# B&R Automation Studio project BenchEDM_AS6
Automation Studio 6.3.2.2; technology packages: mappCockpit 6.2.1, mappConnect 6.1.0, mappControl 6.1.0, mappMotion 6.2.0, mappSafety 6.2.0, mappServices 6.2.0, mappView 6.2.0, OpcUaCs 6.0.0

## Configuration Config1

CPU 5APC3100.KBU2-000, AutomationRuntime 6.3.4, Build 11.3.0, Vc 6.0.0

CPU 5PPC2200.AL04-000, AutomationRuntime 6.3.4, Build 11.3.0, Vc 6.0.0

### Task classes (Cpu.sw)
```
Cyclic#1 (cycle 2000 us, tolerance 0 us):
  Sim <- Process.Sim.prg
  InputMan <- Process.InputMan.prg
  Monitor <- Process.Monitor.prg
  Seq_MASTER <- Process.Seq_MASTER.prg
  OutputMan <- Process.OutputMan.prg
Cyclic#8 (cycle 2000 us):
  BuildVer <- BuildVersion.BuildVer.prg
  Services <- Services.prg
  Vis <- Vis.prg
  Dev <- Dev.prg
DataObjects: MbRTU <- Libraries.MbRTU.dob, McAcpSys, datamod
NcDataObjects: AcpParTabL <- Libraries.AcpParTabL.dob, McDriveLog
Binaries: udbdef, mvLoader, TCLang, TCData, FWRules, ArSvcReg, mvConfig, McAcpSim, McAcpDrv, McMechSys, mvDatApi, McProfGen, BRRole, iomap, asfw, Role, ashwac, UaCsConfig, sysconf, TC, ashwd, User, arconfig, AlarmHist, Config, AlarmCore, AlarmList, Config_1, mCoWebSc, Settings, Config_2, Hierarchy, Config_3, Config_4, Config_6, asnxdb1, Config_5, AlarmCat
ReActionTechnologyObjects: StepDir <- StepDir.prg
Libraries: TC_General, TC_Version, TC_IO, TC_Dir, TC_Convert, TC_ItemX, TC_Array, TC_SysErr, TC_Eval, TC_Mon, TC_Recipe, TC_Sim, TC_AlarmX, TC_RAND, operator, runtime, AsIecCon, astime, ArEventLog, ArProject, AsBrStr, brsystem, FileIO, AsUSB, standard, ArTextSys, sys_lib, MTTypes, MTBasics, MTFilter, AsSMTP, ArCert, ArSsl, AsIODiag, AsTCP, AsXml, MpAlarmX, MpBase, MpRecipe, McBase, MpAxis, McAxis, McAcpAx, AsZip, McAxGroup, McPathGen, McProgInt, SfDomain, MpCnc, McPureVAx, AsIORTI, TC_Str, CoTrace, DRV_mbus, dvframe, DataObj, HA_Matrix, TC_NGRC, TC_Seq, TC_JSON, AsBrMath, TC_FrSky, AsUDP, UaCoal, UaCoalPrv, powerlnk, AsEPL, SfDomDrv, AsIO, AsMem, AsIOAcc, ArUser, MpSfDomMgr, SfDomVis, AsArProf
```

### Hardware
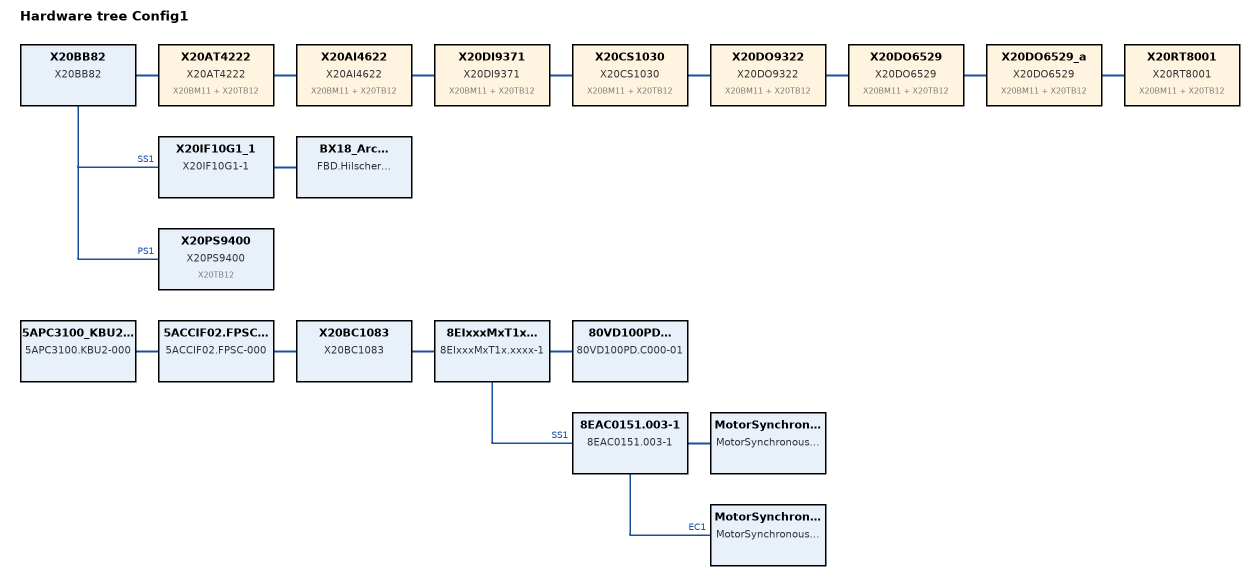
```
5ACCIF02.FPSC-000_a : 5ACCIF02.FPSC-000 v1.6.0.0  [SL -> 5APC3100_KBU2_000_a.SL2]
  Connector IF1:
    EplNatSubnet = 192.168.102.0
    Channel1
    ChannelID1 = McAcpBroadcast
    ChannelType1 = OCTET[96]
  Supervision = off
5APC3100_KBU2_000_a : 5APC3100.KBU2-000 v2.3.0.0
  Connector IF3:
    AssignedOperatingSystem = GPOS
  Connector IF4:
    AssignedOperatingSystem = ARemb
    ActivateDevice = 1
    Mode = Manual
    InternetAddress = 192.168.0.2
    SubnetMask = 255.255.255.0
    ActivateSnmp = 2
  Connector IF9:
    OperatingSystem = ARemb
    ActivateDevice = 1
  Connector IF5:
    AssignedOperatingSystem = GPOS
  Connector IF6:
    AssignedOperatingSystem = GPOS
  Connector IF7:
    AssignedOperatingSystem = ARemb
  Connector IF8:
    AssignedOperatingSystem = ARemb
  ConfigurationID = Config1
  UserPartitionSize = 10000
  UserRamDevice = PCI.2.FPSC.SRAM
  UserRamSize = 14000
  RemMemDevice = PCI.2.FPSC.SRAM
  RemMemSize = 200000
  RemanentGlobalPvSize = 200000
  VolatileGlobalPvSize = 6553500
  ClearNvMemoryAfterShutdownFlushError = 0
  CyclicFlushRemMemSelector = 1
  CyclicFlushRemMemCycleTime = 300
  EnableUsbRemoteInstall = 1
  TimerDeviceType = EPLX2X
  TimerDevice = 5ACCIF02.FPSC-000_a.IF1
  TaskClassIdleTime = 10000
  Cyclic1Duration = 2000
  Cyclic1Tolerance = 0
  Cyclic1Stack = 655360
  Cyclic1Output = 1
  Cyclic8Duration = 2000
  FileDevice1
  FileDeviceName1 = USER_DEVICE
  FileDevicePath1 = F:\
  FileDevice2
  FileDeviceName2 = USER_DEVICE_SIM
  FileDevicePath2 = ..\..\..\..\USER_DEVICE\
  EthernetDefaultGateway = 192.168.0.1
  ActivateFtpServer = 1
  FTPProtocol = 1
  FtpUser1
  FtpUsername1 = brcpu
  FtpUserPassword1 = Ga9FbfaYwFdrzzlreMI/KhLrdRli8oqxPKsqgG5NU/A=
  FtpUserSalt1 = BqJHaXjm
  FTPAccessRight1 = 0
  FTPdevice1 = ALL
  ActivateWebServer = 1
  WebServerProtocol = 1
  ActivateSdm = 1
  ActivateHypervisor = 1
  ARembDramSizeInMb = 3072
80VD100PD.C000-01 : 80VD100PD.C000-01 v2.5.1.0 (NodeNumber=3)  [PLK1 -> 8EIxxxMxT1x.xxxx-1.PLK2 [Cable Type=PowerlinkCable, Length=10, Version=1.0.0.3]]
  DriveConfiguration/Channel[1]/RealAxis:
    AxisReference = gAxisRV_0_0
  DriveConfiguration/Channel[1]/RealAxis/MechanicalElements/Gearbox:
    Input = 10
  DriveConfiguration/Channel[1]/RealAxis/Controller/Mode/Position:
    IntegrationTime = 0.05
  DriveConfiguration/Channel[1]/RealAxis/Controller/Mode/Speed:
    ProportionalGain = 0.2
  DriveConfiguration/Channel[1]/RealAxis/MovementErrorLimits:
    VelocityErrorMonitoring = NotUsed
  DriveConfiguration/Channel[1]/RealAxis/DigitalInputs/Quickstop:
    Input = NotUsed
  DriveConfiguration/Channel[1]/ChannelFeatures:
    FeatureRef[1] = Feature_AcpParTable
  DriveConfiguration/Channel[2]/RealAxis:
    AxisReference = gAxisRT_0_0
  DriveConfiguration/Channel[2]/RealAxis/Controller/Mode/Position:
    ProportionalGain = 500
    IntegrationTime = 0.01
    PredictionTime = 0.003
    TotalDelayTime = 0.003
  DriveConfiguration/Channel[2]/RealAxis/Controller/Mode/Speed:
    ProportionalGain = 0.05
  DriveConfiguration/Channel[2]/RealAxis/MovementErrorLimits:
    VelocityErrorMonitoring = NotUsed
  DriveConfiguration/Channel[2]/RealAxis/DigitalInputs/Quickstop:
    Input = NotUsed
  DriveConfiguration/Channel[2]/ChannelFeatures:
    FeatureRef[1] = Feature_AcpParTable
8EAC0151.003-1 : 8EAC0151.003-1 v2.2.1.0  [SS -> 8EIxxxMxT1x.xxxx-1.SS1; EC1 -> MotorSynchronous_any_a.EC; EC2 -> MotorSynchronous_any.EC]
  Encoder/EncoderX41x:
    InterfaceType = IncrementalEAC151
  Encoder/EncoderX41x/InterfaceType/PowerSupply:
    ReferencePulseDetection = 512
    LineCount = 5000
  Encoder/EncoderX42x:
    InterfaceType = IncrementalEAC151
  Encoder/EncoderX42x/InterfaceType/PowerSupply:
    ReferencePulseDetection = 512
    LineCount = 5000
8EIxxxMxT1x.xxxx-1 : 8EIxxxMxT1x.xxxx-1 v2.4.0.0 (NodeNumber=2)  [PLK1 -> X20BC1083.PLK2 [Cable Type=PowerlinkCable, Length=10, Version=1.0.0.3]; PLK2 -> 80VD100PD.C000-01.PLK1 [Cable Type=PowerlinkCable, Length=10, Version=1.0.0.3]; MT2 -> MotorSynchronous_any.MT]
  PDMConfig = DoubleAxis
  DriveConfiguration/Encoder/EncoderX43:
    InterfaceType = EnDat
  DriveConfiguration/Channel[1]/RealAxis:
    AxisReference = gAxisRY_0_0
  DriveConfiguration/Channel[1]/RealAxis/MechanicalElements/RotaryToLinearTransformation:
    ReferenceDistance = 20
  DriveConfiguration/Channel[1]/RealAxis/EncoderLink:
    MotorAndPositionEncoder = EncoderX41x
  DriveConfiguration/Channel[1]/RealAxis/Controller:
    Mode = PositionControllerWithTorqueFeedForward
  DriveConfiguration/Channel[1]/RealAxis/Controller/Mode/Position:
    ProportionalGain = 500
    IntegrationTime = 0.1
  DriveConfiguration/Channel[1]/RealAxis/Controller/Mode/Speed:
    ProportionalGain = 0.5
  DriveConfiguration/Channel[1]/RealAxis/Controller/Mode/FeedForward:
    TorquePositive = 0.2
    TorqueNegative = 0.2
    SpeedTorqueFactor = 0.005
    Inertia = 0.00015
  DriveConfiguration/Channel[1]/RealAxis/Homing:
    Mode = BlockTorque
  DriveConfiguration/Channel[1]/RealAxis/Homing/Mode:
    Position = -20
    StartVelocity = 20
    HomingVelocity = 20
    Acceleration = 1000
    StartDirection = Negative
    TorqueLimit = 1.5
    PositionErrorStopLimit = 4
  DriveConfiguration/Channel[1]/RealAxis/MovementErrorLimits:
    PositionError = 5
    VelocityErrorMonitoring = NotUsed
  DriveConfiguration/Channel[1]/ChannelFeatures:
    FeatureRef[1] = Feature_AcpParTable
  DriveConfiguration/Channel[2]/RealAxis:
    AxisReference = gAxisRX_0_0
  DriveConfiguration/Channel[2]/RealAxis/MechanicalElements/RotaryToLinearTransformation:
    ReferenceDistance = 20
  DriveConfiguration/Channel[2]/RealAxis/EncoderLink:
    MotorAndPositionEncoder = EncoderX42x
  DriveConfiguration/Channel[2]/RealAxis/Controller/Mode/Position:
    ProportionalGain = 500
    IntegrationTime = 0.1
  DriveConfiguration/Channel[2]/RealAxis/Controller/Mode/Speed:
    ProportionalGain = 0.5
  DriveConfiguration/Channel[2]/RealAxis/Homing:
    Mode = BlockTorque
  DriveConfiguration/Channel[2]/RealAxis/Homing/Mode:
    Position = -10
    StartVelocity = 20
    HomingVelocity = 20
    Acceleration = 1000
    StartDirection = Negative
    TorqueLimit = 1.5
    PositionErrorStopLimit = 4
  DriveConfiguration/Channel[2]/RealAxis/MovementErrorLimits:
    PositionError = 5
    VelocityErrorMonitoring = NotUsed
  DriveConfiguration/Channel[2]/ChannelFeatures:
    FeatureRef[1] = Feature_AcpParTable
  DriveConfiguration/Channel[3]/RealAxis:
    AxisReference = 
BX18_Arc_Generator_V1_0 : FBD.Hilscher.ECATGenSlaveDTM.BX18 Arc Generator V1.0 v1.0 (OrderNumber=BX18 Arc Generator V1.0)  [ECAT1 -> X20IF10G1_1.IF1]
  DtmId = 61a48d3a-efc3-4167-a8a5-4e7e0e28ba40
MotorSynchronous_any : MotorSynchronous_any v2.2.1.0  [EC -> 8EAC0151.003-1.EC2; MT -> 8EIxxxMxT1x.xxxx-1.MT2]
  M1/MotorParameters:
    MOTOR_POLEPAIRS = 1
    MOTOR_SPEED_RATED = 3300
    MOTOR_SPEED_MAX = 9300
    MOTOR_VOLTAGE_RATED = 300
    MOTOR_CURR_RATED = 2
    MOTOR_CURR_STALL = 2
    MOTOR_CURR_MAX = 8
    MOTOR_TORQ_RATED = 0.66
    MOTOR_TORQ_STALL = 2.55
    MOTOR_TORQ_MAX = 2.65
    MOTOR_VOLTAGE_CONST = 10.53
    MOTOR_TORQ_CONST = 0.302
    MOTOR_STATOR_RESISTANCE = 1.3
    MOTOR_STATOR_INDUCTANCE = 3.8
    MOTOR_INERTIA = 0.172
  M1/MotorParameters/EncoderMounting:
    Angle = Undefined
  M1/MotorParameters/EncoderMounting/Angle:
    AutomaticIdentification = Dither
  M1/MotorParameters/EncoderMounting/Angle/AutomaticIdentification:
    PHASING_CURR = 1.5 (Disabled=false)
  M1/MotorParameters:
    TemperatureSensor = NotUsed
    TemperatureModel = NotUsed
MotorSynchronous_any_a : MotorSynchronous_any v2.2.1.0  [EC -> 8EAC0151.003-1.EC1; MT -> 8EIxxxMxT1x.xxxx-1.MT1]
  M1/MotorParameters:
    MOTOR_POLEPAIRS = 1
    MOTOR_SPEED_RATED = 3300
    MOTOR_SPEED_MAX = 9300
    MOTOR_VOLTAGE_RATED = 300
    MOTOR_CURR_RATED = 2
    MOTOR_CURR_STALL = 2
    MOTOR_CURR_MAX = 8
    MOTOR_TORQ_RATED = 0.66
    MOTOR_TORQ_STALL = 2.55
    MOTOR_TORQ_MAX = 2.65
    MOTOR_VOLTAGE_CONST = 10.53
    MOTOR_TORQ_CONST = 0.302
    MOTOR_STATOR_RESISTANCE = 1.3
    MOTOR_STATOR_INDUCTANCE = 3.8
    MOTOR_INERTIA = 0.172
  M1/MotorParameters/EncoderMounting:
    Angle = Undefined
  M1/MotorParameters/EncoderMounting/Angle:
    AutomaticIdentification = Dither
  M1/MotorParameters/EncoderMounting/Angle/AutomaticIdentification:
    PHASING_CURR = 1.5 (Disabled=false)
  M1/MotorParameters:
    TemperatureSensor = NotUsed
    TemperatureModel = NotUsed
X20AI4622 : X20AI4622 v1.5.0.0  [SS1 -> X20TB12_c.SS; SL -> X20BM11_b.SL1]
  Supervision = off
  ChannelType01 = 0 to 20mA
  ChannelType02 = 0 to 20mA
  ChannelType03 = 0 to 20mA
  ChannelType04 = 0 to 20mA
X20AT4222 : X20AT4222 v1.6.2.0  [SS1 -> X20TB12.SS; SL -> X20BM11_a.SL1]
  Supervision = off
X20BB82 : X20BB82 v1.2.0.0
X20BC1083 : X20BC1083 v2.16.1.0 (NodeNumber=1)  [PLK1 -> 5ACCIF02.FPSC-000_a.IF1 [Cable Type=PowerlinkCable, Length=10, Version=1.0.0.3]; PLK2 -> 8EIxxxMxT1x.xxxx-1.PLK1 [Cable Type=PowerlinkCable, Length=10, Version=1.0.0.3]; SL -> X20BB82.SL1]
  Supervision = off
X20BM11 : X20BM11 v1.1.0.0  [X2X1 -> X20BM11_g.X2X2]
X20BM11_a : X20BM11 v1.1.0.0  [X2X1 -> X20BB82.IF1]
X20BM11_b : X20BM11 v1.1.0.0  [X2X1 -> X20BM11_a.X2X2]
X20BM11_c : X20BM11 v1.1.0.0  [X2X1 -> X20BM11_b.X2X2]
X20BM11_d : X20BM11 v1.1.0.0  [X2X1 -> X20BM11_c.X2X2]
X20BM11_e : X20BM11 v1.1.0.0  [X2X1 -> X20BM11_d.X2X2]
X20BM11_f : X20BM11 v1.1.0.0  [X2X1 -> X20BM11_e.X2X2]
X20BM11_g : X20BM11 v1.1.0.0  [X2X1 -> X20BM11_f.X2X2]
X20CS1030 : X20CS1030 v1.8.3.0  [SS1 -> X20TB12_e.SS; SL -> X20BM11_d.SL1]
  Supervision = off
X20DI9371 : X20DI9371 v1.6.1.0  [SS1 -> X20TB12_d.SS; SL -> X20BM11_c.SL1]
  Supervision = off
X20DO6529 : X20DO6529 v1.4.1.0  [SS1 -> X20TB12_g.SS; SL -> X20BM11_f.SL1]
  Supervision = off
X20DO6529_a : X20DO6529 v1.4.1.0  [SS1 -> X20TB12_h.SS; SL -> X20BM11_g.SL1]
  Supervision = off
X20DO9322 : X20DO9322 v1.7.0.0  [SS1 -> X20TB12_f.SS; SL -> X20BM11_e.SL1]
  Supervision = off
X20IF10G1_1 : X20IF10G1-1 v1.0.2.0  [SS -> X20BB82.SS1]
  Connector IF1:
    DtmRef = FBDIF.Hilscher.ECATMasterDTM.NETX 100 RE/ECM
    DtmId = 2adc853f-087f-4c82-9441-944b4b0f2f89
  ConfigFile = X20IF10G1_1.dtm
  ConfigModule = asnxdb1
  CycleTime = 2000
X20PS9400 : X20PS9400 v1.8.1.0  [SS1 -> X20TB12_b.SS; PS -> X20BB82.PS1]
  Supervision = off
X20RT8001 : X20RT8001 v1.7.2.0  [SS1 -> X20TB12_a.SS; SL -> X20BM11.SL1]
  Supervision = off
  ReActionTask = StepDir
  ReActionTaskDisabled = FALSE
  TypePar1 = DINT
  TypePar2 = DINT
  TypePar3 = DINT
  TypeRes1 = DINT
X20TB12 : X20TB12 v1.0.0.0
X20TB12_a : X20TB12 v1.0.0.0
X20TB12_b : X20TB12 v1.0.0.0
X20TB12_c : X20TB12 v1.0.0.0
X20TB12_d : X20TB12 v1.0.0.0
X20TB12_e : X20TB12 v1.0.0.0
X20TB12_f : X20TB12 v1.0.0.0
X20TB12_g : X20TB12 v1.0.0.0
X20TB12_h : X20TB12 v1.0.0.0
```

### IoMap.iom - 5APC3100_KBU2_000_a/IoMap.iom
```iecst
VAR_CONFIG
	Cyclic#1.gIO.BX18.Outputs_control AT %QW."BX18_Arc_Generator_V1_0".Outputs_control;
	Cyclic#1.gIO.BX18.Outputs_onTime AT %QW."BX18_Arc_Generator_V1_0".Outputs_onTime;
	Cyclic#1.gIO.BX18.Outputs_offTime AT %QW."BX18_Arc_Generator_V1_0".Outputs_offTime;
	Cyclic#1.gIO.BX18.Outputs_current AT %QW."BX18_Arc_Generator_V1_0".Outputs_current;
	Cyclic#1.gIO.BX18.Inputs_status AT %IW."BX18_Arc_Generator_V1_0".Inputs_status;
	Cyclic#1.gIO.BX18.Inputs_EDMservofeedback AT %IW."BX18_Arc_Generator_V1_0".Inputs_EDMservofeedback;
	Cyclic#1.gIO.BX18.Inputs_power AT %IW."BX18_Arc_Generator_V1_0".Inputs_power;
	Cyclic#1.gIO.BX18.ModuleOK AT %IX."BX18_Arc_Generator_V1_0".ModuleOk;
	Cyclic#1.::gIO.Motion.ModuleOK AT %IX."X20RT8001".ModuleOk;
	Cyclic#1.::gIO.Motion.ENABLED AT %IX."X20RT8001".RTEngineRun;
	Cyclic#1.::gIO.Motion.ActualPosition AT %ID."X20RT8001".RES01;
	Cyclic#1.::gIO.Motion.SetPosition AT %QD."X20RT8001".PAR01;
	Cyclic#1.::gIO.Motion.Home AT %QD."X20RT8001".PAR02;
	Cyclic#1.::gIO.Motion.ENABLE AT %QX."X20RT8001".RTEnable;
	Cyclic#1.::gIO.Safety.TC_IO_DI_ESTOP.IOMapping AT %IX."X20DI9371".DigitalInput01;
	Cyclic#1.::gIO.Motion.StepDelay AT %QD."X20RT8001".PAR03;
	Cyclic#1.::gIO.Motion.TC_IO_DI_HomeSwitchZ.IOMapping AT %IX."X20DI9371".DigitalInput03;
END_VAR
```

### Config.mappconnect - 5APC3100_KBU2_000_a/mappConnect/Config.mappconnect
```
Element mapp Connect Configuration (Type=mappconnect)
  WebServerProtocol = 1
    WebServerPort = 8081
    Interface = All
    WebServerPortSsl = 8443
  WebServerEndpointConfiguration:
    Endpoint[1]:
      Endpoint = *.*
      Roles
  OpcUaServerWhitelist:
    OpcUaServer[1]:
      Url = opc.tcp://127.0.0.1:4840
```

### Config_1.axesgroup - 5APC3100_KBU2_000_a/mappMotion/CNC/Config_1.axesgroup
```
Element gCNC (Type=axesgroup)
  Type = PathGenAxesGroup
    PhysicalAxes:
      JointAxes:
        JointAxis[1]:
          Name = QX
          AxisRef = gAxisVX_0
        JointAxis[2]:
          Name = QY
          AxisRef = gAxisVY_0
        JointAxis[3]:
          Name = QZ
          AxisRef = gAxisVZ_0
    MechanicalSystem:
      MechSysRef = MechSys
    AxesGroupFeatures:
      FeatureRef[1] = Feature_Programs
      FeatureRef[2] = Feature_ReverseMovement
  Alarms = MpAlarmX
```

### Config_2.axis - 5APC3100_KBU2_000_a/mappMotion/CNC/Config_2.axis
```
Element gAxisRP_1_0 (Type=axis)
  BaseType:
    MeasurementUnit = 5059636
    MeasurementResolution = 0.001
    PeriodSettings:
      Period = 1
  MovementLimits:
    Velocity:
      Velocity = 60
    Acceleration:
      Acceleration = 600
    Deceleration:
      Deceleration = 600
  Alarms = MpAlarmX
Element gAxisRP_0_0 (Type=axis)
  BaseType:
    MeasurementUnit = 5059636
    MeasurementResolution = 0.001
    PeriodSettings:
      Period = 1
  MovementLimits:
    Velocity:
      Velocity = 60
    Acceleration:
      Acceleration = 600
    Deceleration:
      Deceleration = 600
  Alarms = MpAlarmX
Element gAxisRT_0_0 (Type=axis)
  BaseType:
    MeasurementResolution = 0.001
  MovementLimits:
    Velocity:
      Velocity = 12000
    Acceleration:
      Acceleration = 120000
    Deceleration:
      Deceleration = 120000
  Alarms = MpAlarmX
Element gAxisRV_0_0 (Type=axis)
  BaseType:
    MeasurementResolution = 0.001
  MovementLimits:
    Velocity:
      Velocity = 1200
    Acceleration:
      Acceleration = 12000
    Deceleration:
      Deceleration = 12000
  Alarms = MpAlarmX
Element gAxisRX_0_0 (Type=axis)
  BaseType = LinearBounded
    MeasurementResolution = 0.001
  MovementLimits:
    Position:
      LowerLimit = 0
      UpperLimit = 250
    Velocity:
      Velocity = 1000
    Acceleration:
      Acceleration = 5000
    Deceleration:
      Deceleration = 5000
  Alarms = MpAlarmX
Element gAxisRY_0_0 (Type=axis)
  BaseType = LinearBounded
    MeasurementResolution = 0.001
  MovementLimits:
    Position:
      LowerLimit = 0
      UpperLimit = 550
    Velocity:
      Velocity = 1000
    Acceleration:
      Acceleration = 5000
    Deceleration:
      Deceleration = 5000
  Alarms = MpAlarmX
Element gAxisRZ_0_0 (Type=axis)
  BaseType = LinearBounded
    MeasurementResolution = 0.001
  MovementLimits:
    Position:
      LowerLimit = 0
      UpperLimit = 265
    Velocity:
      Velocity = 120
    Acceleration:
      Acceleration = 12000
    Deceleration:
      Deceleration = 12000
  Alarms = MpAlarmX
Element gAxisVT_0 (Type=axis)
  BaseType:
    MeasurementResolution = 0.001
  MovementLimits:
    Velocity:
      Velocity = 10000
    Acceleration:
      Acceleration = 100000
    Deceleration:
      Deceleration = 100000
  Alarms = MpAlarmX
Element gAxisVV_0 (Type=axis)
  BaseType:
    MeasurementResolution = 0.001
  MovementLimits:
    Velocity:
      Velocity = 1000
    Acceleration:
      Acceleration = 10000
    Deceleration:
      Deceleration = 10000
  Alarms = MpAlarmX
Element gAxisVX_0 (Type=axis)
  BaseType = LinearBounded
    MeasurementResolution = 0.001
  MovementLimits:
    Position:
      LowerLimit = 0
      UpperLimit = 250
    Velocity:
      Velocity = 800
    Acceleration:
      Acceleration = 4000
    Deceleration:
      Deceleration = 4000
  Alarms = MpAlarmX
Element gAxisVY_0 (Type=axis)
  BaseType = LinearBounded
    MeasurementResolution = 0.001
  MovementLimits:
    Position:
      LowerLimit = 0
      UpperLimit = 550
    Velocity:
      Velocity = 800
    Acceleration:
      Acceleration = 4000
    Deceleration:
      Deceleration = 4000
  Alarms = MpAlarmX
Element gAxisVZ_0 (Type=axis)
  BaseType = LinearBounded
    MeasurementResolution = 0.001
  MovementLimits:
    Position:
      LowerLimit = 0
      UpperLimit = 265
    Velocity:
      Velocity = 100
    Acceleration:
      Acceleration = 10000
    Deceleration:
      Deceleration = 10000
  Alarms = MpAlarmX
```

### Config_3.mechanicalsystem - 5APC3100_KBU2_000_a/mappMotion/CNC/Config_3.mechanicalsystem
```
Element MechSys (Type=mechanicalsystem)
  Type = 3AxesCNC
    Subtype:
      JointAxesPositionLimits:
        JointAxis[1]
        JointAxis[2]
        JointAxis[3]
```

### Config_4.axesgroupfeature - 5APC3100_KBU2_000_a/mappMotion/CNC/Config_4.axesgroupfeature
```
Element Feature_Programs (Type=axesgroupfeature)
  Type:
    Location = User
      UserLocation[1]:
        FileDevice = USER_DEVICE
      UserLocation[2]:
        FileDevice = USER_DEVICE_SIM
Element Feature_ReverseMovement (Type=axesgroupfeature)
  Type = ReverseMovement
    Distance = 5
```

### Config_5.purevaxcfg - 5APC3100_KBU2_000_a/mappMotion/CNC/Config_5.purevaxcfg
```
Element PureVAxCfg_VT_0 (Type=purevaxcfg)
  PureVAxis:
    AxisReference = gAxisVT_0
Element PureVAxCfg_VV_0 (Type=purevaxcfg)
  PureVAxis:
    AxisReference = gAxisVV_0
Element PureVAxCfg_RZ_0_0 (Type=purevaxcfg)
  PureVAxis:
    AxisReference = gAxisRZ_0_0
    Homing:
      Mode = LimitSwitch
        Position = -5
        StartVelocity = 20
        HomingVelocity = 5
        Acceleration = 12000
        SwitchEdge = Negative
    GeneralPurposeAxisInterface = Used
      MovementErrorLimits:
        PositionError = 1000
      DigitalInputs:
        NegativeLimitSwitch:
          Source = InputPV
            PVmapping = gIO.Motion.TC_IO_DI_HomeSwitchZ.Signal.Filtered
        Trigger1:
          Source = InputPV
            PVmapping = ::gIO.Safety.TC_IO_DI_ESTOP.Signal.Filtered
          Level = Low
        Quickstop:
          Input = Trigger1
      StatusInputs:
        PoweredOn:
          Source = InputPV
            PVmapping = ::gIO.Motion.SwitchedOn
        ReadyForPowerOn:
          Source = InputPV
            PVmapping = ::gIO.Motion.ENABLED
      ControlOutputs:
        PowerOn = Used
          Destination:
            PVmapping = ::gIO.Motion.SwitchOn
Element PureVAxCfg_VZ_0 (Type=purevaxcfg)
  PureVAxis:
    AxisReference = gAxisVZ_0
Element PureVAxCfg_VY_0 (Type=purevaxcfg)
  PureVAxis:
    AxisReference = gAxisVY_0
Element PureVAxCfg_VX_0 (Type=purevaxcfg)
  PureVAxis:
    AxisReference = gAxisVX_0
Element PureVAxCfg_RP_1_0 (Type=purevaxcfg)
  PureVAxis:
    AxisReference = gAxisRP_1_0
    GeneralPurposeAxisInterface = DS402VL
      MovementErrorLimits:
        PositionError = 10
      VelocityActualValue:
        Source = Variable
          PVMapping = ::gIO.VFD[1].RFRD
      StatusInputs:
        StatusWord:
          Source = InputPV
            PVmapping = ::gIO.VFD[1].ETA
      ControlOutputs:
        ControlWord:
          Destination:
            PVMapping = ::gIO.VFD[1].CMD
        TargetVelocity:
          Destination:
            PVmapping = ::gIO.VFD[1].LFRD
Element PureVAxCfg_RP_0_0 (Type=purevaxcfg)
  PureVAxis:
    AxisReference = gAxisRP_0_0
    GeneralPurposeAxisInterface = DS402VL
      MovementErrorLimits:
        PositionError = 10
      VelocityActualValue:
        Source = Variable
          PVMapping = ::gIO.VFD[0].RFRD
      StatusInputs:
        StatusWord:
          Source = InputPV
            PVmapping = ::gIO.VFD[0].ETA
      ControlOutputs:
        ControlWord:
          Destination:
            PVMapping = ::gIO.VFD[0].CMD
        TargetVelocity:
          Destination:
            PVmapping = ::gIO.VFD[0].LFRD
```

### Config_6.axisfeature - 5APC3100_KBU2_000_a/mappMotion/CNC/Config_6.axisfeature
```
Element Feature_AcpParTable (Type=axisfeature)
  Type = ParTab
    ParTabRef = AcpParTabL
```

### AlarmList.mpalarmxlist - 5APC3100_KBU2_000_a/mappServices/AlarmList.mpalarmxlist
```
Element gAlarmXList_Base (Type=mpalarmxlist)
  mapp.AlarmX.Core.Configuration:
    [0]:
      Name = {1}Severity0
      Message = {$IAT/Alarm.{1}Severity}
      Code = 0
      Severity = 0
      Behavior = EdgeAlarm
        Confirm = 0
        ReactionWhilePending = TRUE
        Retain = FALSE
        Async = FALSE
        DataUpdate:
          Activation:
            TimeStamp = FALSE
            Snippets = FALSE
        Recording:
          InactiveToActive = TRUE
          UnacknowledgedToAcknowledged = FALSE
          AcknowledgedToUnacknowledged = FALSE
          UnconfirmedToConfirmed = FALSE
          ConfirmedToUnconfirmed = FALSE
      Disable = FALSE
      InhibitPV
      AdditionalInformation1
      AdditionalInformation2
    [1]:
      Name = {1}Severity1
      Message = {$IAT/Alarm.{1}Severity}
      Code = 1
      Severity = 1
      Behavior = EdgeAlarm
        Confirm = 0
        ReactionWhilePending = TRUE
        Retain = FALSE
        Async = FALSE
        DataUpdate:
          Activation:
            TimeStamp = FALSE
            Snippets = FALSE
        Recording:
          InactiveToActive = TRUE
          UnacknowledgedToAcknowledged = FALSE
          AcknowledgedToUnacknowledged = FALSE
          UnconfirmedToConfirmed = FALSE
          ConfirmedToUnconfirmed = FALSE
      Disable = FALSE
      InhibitPV
      AdditionalInformation1
      AdditionalInformation2
    [2]:
      Name = {1}Severity2
      Message = {$IAT/Alarm.{1}Severity}
      Code = 2
      Severity = 2
      Behavior = EdgeAlarm
        Confirm = 0
        ReactionWhilePending = TRUE
        Retain = FALSE
        Async = FALSE
        DataUpdate:
          Activation:
            TimeStamp = FALSE
            Snippets = FALSE
        Recording:
          InactiveToActive = TRUE
          UnacknowledgedToAcknowledged = FALSE
          AcknowledgedToUnacknowledged = FALSE
          UnconfirmedToConfirmed = FALSE
          ConfirmedToUnconfirmed = FALSE
      Disable = FALSE
      InhibitPV
      AdditionalInformation1
      AdditionalInformation2
    [3]:
      Name = {1}Severity3
      Message = {$IAT/Alarm.{1}Severity}
      Code = 3
      Severity = 3
      Behavior = EdgeAlarm
        Confirm = 0
        ReactionWhilePending = TRUE
        Retain = FALSE
        Async = FALSE
        DataUpdate:
          Activation:
            TimeStamp = FALSE
            Snippets = FALSE
        Recording:
          InactiveToActive = TRUE
          UnacknowledgedToAcknowledged = FALSE
          AcknowledgedToUnacknowledged = FALSE
          UnconfirmedToConfirmed = FALSE
          ConfirmedToUnconfirmed = FALSE
      Disable = FALSE
      InhibitPV
      AdditionalInformation1
      AdditionalInformation2
    [4]:
      Name = {1}Severity4
      Message = {$IAT/Alarm.{1}Severity}
      Code = 4
      Severity = 4
      Behavior = EdgeAlarm
        Confirm = 0
        ReactionWhilePending = TRUE
        Retain = FALSE
        Async = FALSE
        DataUpdate:
          Activation:
            TimeStamp = FALSE
            Snippets = FALSE
        Recording:
          InactiveToActive = TRUE
          UnacknowledgedToAcknowledged = FALSE
          AcknowledgedToUnacknowledged = FALSE
          UnconfirmedToConfirmed = FALSE
          ConfirmedToUnconfirmed = FALSE
      Disable = FALSE
      InhibitPV
      AdditionalInformation1
      AdditionalInformation2
  mapp.AlarmX.Snippets:
    AutoDetect = 1
      Language
    [0]:
      Key = TestKey
      Value = PV
        PV = ::gRem.RuntimeHours
      Alarm
```

### Config_1.axesgroup - 5PPC2200_AL04_000/mappMotion/CNC/Config_1.axesgroup
```
Element gCNC (Type=axesgroup)
  Type = PathGenAxesGroup
    PhysicalAxes:
      JointAxes:
        JointAxis[1]:
          Name = QX
          AxisRef = gAxisVX_0
        JointAxis[2]:
          Name = QY
          AxisRef = gAxisVY_0
        JointAxis[3]:
          Name = QZ
          AxisRef = gAxisVZ_0
      SlaveAxes:
        SlaveAxis[1]:
          Name = QT
          AxisRef = gAxisVT_0
        SlaveAxis[2]:
          Name = QV
          AxisRef = gAxisVV_0
    MechanicalSystem:
      MechSysRef = MechSys
    AxesGroupFeatures:
      FeatureRef[1] = Feature_Programs
  Alarms = MpAlarmX
```

### Config_4.axesgroupfeature - 5PPC2200_AL04_000/mappMotion/CNC/Config_4.axesgroupfeature
```
Element Feature_Programs (Type=axesgroupfeature)
  Type:
    Location = User
      UserLocation[1]:
        FileDevice = USER_DEVICE
      UserLocation[2]:
        FileDevice = USER_DEVICE_SIM
```

### Config_5.purevaxcfg - 5PPC2200_AL04_000/mappMotion/CNC/Config_5.purevaxcfg
```
Element PureVAxCfg_VT_0 (Type=purevaxcfg)
  PureVAxis:
    AxisReference = gAxisVT_0
Element PureVAxCfg_VV_0 (Type=purevaxcfg)
  PureVAxis:
    AxisReference = gAxisVV_0
Element PureVAxCfg_RZ0_0 (Type=purevaxcfg)
  PureVAxis:
    AxisReference = gAxisRZ0_0
Element PureVAxCfg_VZ_0 (Type=purevaxcfg)
  PureVAxis:
    AxisReference = gAxisVZ_0
Element PureVAxCfg_VY_0 (Type=purevaxcfg)
  PureVAxis:
    AxisReference = gAxisVY_0
Element PureVAxCfg_VX_0 (Type=purevaxcfg)
  PureVAxis:
    AxisReference = gAxisVX_0
```

### AlarmCore.mpalarmxcore - 5PPC2200_AL04_000/mappServices/AlarmCore.mpalarmxcore
```
Element gAlarmXCore (Type=mpalarmxcore)
  mapp.Gen:
    Enable = TRUE
    EnableCockpit = TRUE
    TaskClass = 1
    Parent
  mapp.AlarmX.Core:
    Mapping:
      [0]:
        Alarm = [0..99]
        Action = Reaction
          Name = SeverityAny
      [1]:
        Alarm = [0..0]
        Action = Reaction
          Name = Severity0
      [2]:
        Alarm = [1..1]
        Action = Reaction
          Name = Severity1
      [3]:
        Alarm = [2..2]
        Action = Reaction
          Name = Severity2
      [4]:
        Alarm = [3..3]
        Action = Reaction
          Name = Severity3
      [5]:
        Alarm = [4..4]
        Action = Reaction
          Name = Severity4
  mapp.AlarmX.List:
    [0]:
      List = gAlarmXList_Base
      Offset = 9000
      Argument1 = Monitor
  mapp.AlarmX.Create = Disabled
  mapp.AlarmX.Core.Retain:
    Memory = 0
```

### AlarmHist.mpalarmxhistory - 5PPC2200_AL04_000/mappServices/AlarmHist.mpalarmxhistory
```
Element gAlarmXHistory (Type=mpalarmxhistory)
  mapp.Gen:
    Enable = TRUE
    EnableCockpit = TRUE
    Audit = TRUE
    Parent
  mapp.AlarmX.History:
    Export:
      TimeStampPattern = %Y-%m-%d %H:%M:%S:%L
      AutoExtension = TRUE
      ColumnSeparator = ,
    Memory = 2
      Size = 5
    Scope = 0
```

### Config.mprecipexml - 5PPC2200_AL04_000/mappServices/Config.mprecipexml
```
Element gRecipeXml_Rem (Type=mprecipexml)
  mapp.Gen:
    Enable = TRUE
    EnableCockpit = TRUE
    TaskClass = 8
    Audit = FALSE
    Parent
  mapp.Recipe.Xml:
    AutoSave = Time
      Interval = 600
      StartImmediately = FALSE
    Encryption = FALSE
    PassPhrase
    AutoExtension = TRUE
    Signature = Disabled
  Alarms = MpAlarmX
    mapp.AlarmX.Core.Configuration:
      [0]:
        Name = SaveFailed
        Message = {$BR/mapp/MpRecipeXml/Alarms/SaveFailed}
        Code = 0
        Severity = 1
        Behavior = EdgeAlarm
          AutoReset = TRUE
          Acknowledge = 1
          Confirm = 0
          MultipleInstances = TRUE
          ReactionWhilePending = TRUE
          Async = FALSE
          Recording:
            InactiveToActive = TRUE
            ActiveToInactive = FALSE
            UnacknowledgedToAcknowledged = TRUE
            UnconfirmedToConfirmed = TRUE
        Disable = FALSE
        AdditionalInformation1
        AdditionalInformation2
      [1]:
        Name = SaveFailedPartial
        Message = {$BR/mapp/MpRecipeXml/Alarms/SaveFailedPartial}
        Code = 0
        Severity = 1
        Behavior = EdgeAlarm
          AutoReset = TRUE
          Acknowledge = 1
          Confirm = 0
          MultipleInstances = TRUE
          ReactionWhilePending = TRUE
          Async = FALSE
          Recording:
            InactiveToActive = TRUE
            ActiveToInactive = FALSE
            UnacknowledgedToAcknowledged = TRUE
            UnconfirmedToConfirmed = TRUE
        Disable = FALSE
        AdditionalInformation1
        AdditionalInformation2
      [2]:
        Name = LoadFailed
        Message = {$BR/mapp/MpRecipeXml/Alarms/LoadFailed}
        Code = 0
        Severity = 1
        Behavior = EdgeAlarm
          AutoReset = TRUE
          Acknowledge = 1
          Confirm = 0
          MultipleInstances = TRUE
          ReactionWhilePending = TRUE
          Async = FALSE
          Recording:
            InactiveToActive = TRUE
            ActiveToInactive = FALSE
            UnacknowledgedToAcknowledged = TRUE
            UnconfirmedToConfirmed = TRUE
        Disable = FALSE
        AdditionalInformation1
        AdditionalInformation2
      [3]:
        Name = LoadFailedPartial
        Message = {$BR/mapp/MpRecipeXml/Alarms/LoadFailedPartial}
        Code = 0
        Severity = 1
        Behavior = EdgeAlarm
          AutoReset = TRUE
          Acknowledge = 1
          Confirm = 0
          MultipleInstances = TRUE
          ReactionWhilePending = TRUE
          Async = FALSE
          Recording:
            InactiveToActive = TRUE
            ActiveToInactive = FALSE
            UnacknowledgedToAcknowledged = TRUE
            UnconfirmedToConfirmed = TRUE
        Disable = FALSE
        AdditionalInformation1
        AdditionalInformation2
Element gRecipeXml_Par (Type=mprecipexml)
  mapp.Gen:
    Enable = TRUE
    EnableCockpit = TRUE
    TaskClass = 8
    Audit = FALSE
    Parent
  mapp.Recipe.Xml:
    AutoSave = Standard
    Encryption = FALSE
    PassPhrase
    AutoExtension = TRUE
    Signature = Disabled
  Alarms = MpAlarmX
    mapp.AlarmX.Core.Configuration:
      [0]:
        Name = SaveFailed
        Message = {$BR/mapp/MpRecipeXml/Alarms/SaveFailed}
        Code = 0
        Severity = 1
        Behavior = EdgeAlarm
          AutoReset = TRUE
          Acknowledge = 1
          Confirm = 0
          MultipleInstances = TRUE
          ReactionWhilePending = TRUE
          Async = FALSE
          Recording:
            InactiveToActive = TRUE
            ActiveToInactive = FALSE
            UnacknowledgedToAcknowledged = TRUE
            UnconfirmedToConfirmed = TRUE
        Disable = FALSE
        AdditionalInformation1
        AdditionalInformation2
      [1]:
        Name = SaveFailedPartial
        Message = {$BR/mapp/MpRecipeXml/Alarms/SaveFailedPartial}
        Code = 0
        Severity = 1
        Behavior = EdgeAlarm
          AutoReset = TRUE
          Acknowledge = 1
          Confirm = 0
          MultipleInstances = TRUE
          ReactionWhilePending = TRUE
          Async = FALSE
          Recording:
            InactiveToActive = TRUE
            ActiveToInactive = FALSE
            UnacknowledgedToAcknowledged = TRUE
            UnconfirmedToConfirmed = TRUE
        Disable = FALSE
        AdditionalInformation1
        AdditionalInformation2
      [2]:
        Name = LoadFailed
        Message = {$BR/mapp/MpRecipeXml/Alarms/LoadFailed}
        Code = 0
        Severity = 1
        Behavior = EdgeAlarm
          AutoReset = TRUE
          Acknowledge = 1
          Confirm = 0
          MultipleInstances = TRUE
          ReactionWhilePending = TRUE
          Async = FALSE
          Recording:
            InactiveToActive = TRUE
            ActiveToInactive = FALSE
            UnacknowledgedToAcknowledged = TRUE
            UnconfirmedToConfirmed = TRUE
        Disable = FALSE
        AdditionalInformation1
        AdditionalInformation2
      [3]:
        Name = LoadFailedPartial
        Message = {$BR/mapp/MpRecipeXml/Alarms/LoadFailedPartial}
        Code = 0
        Severity = 1
        Behavior = EdgeAlarm
          AutoReset = TRUE
          Acknowledge = 1
          Confirm = 0
          MultipleInstances = TRUE
          ReactionWhilePending = TRUE
          Async = FALSE
          Recording:
            InactiveToActive = TRUE
            ActiveToInactive = FALSE
            UnacknowledgedToAcknowledged = TRUE
            UnconfirmedToConfirmed = TRUE
        Disable = FALSE
        AdditionalInformation1
        AdditionalInformation2
```

## Logical view

Binary libraries used (declarations not repeated): operator, runtime, AsIecCon, astime, ArEventLog, ArProject, AsBrStr, brsystem, FileIO, AsUSB, standard, ArTextSys, sys_lib, MTTypes, MTBasics 6.1.0, MTFilter 6.1.0, AsSMTP, ArCert, ArSsl, AsIODiag, AsTCP, AsXml, MpAlarmX, MpBase, MpRecipe, McBase, MpAxis, McAxis, McAcpAx, AsZip, McAxGroup, McPathGen, McProgInt, SfDomain, MpCnc 6.2.0, McPureVAx, AsIORTI, CoTrace, DRV_mbus, dvframe, DataObj, AsBrMath, AsUDP

- AutoGenScript.ps1 - Pre-build script (not shown)

### AutoGenMonitor.st
```iecst
{
	MON_SYSTEM_PAR_NOT_READY : {
	  Text: {
	      en: "Parameters NOT Loaded: {&TestKey}",
	      es: "Parámetros No Cargados: {&TestKey}",
	      fr: "Paramètres Non Chargés: {&TestKey}",
	      de: "Parameter Nicht Geladen: {&TestKey}"
	  },
	  Snippets: {
	      TestKey: `gRem.RuntimeHours`,
	  },
	  Sev: 4,
	  Mask: {
	      PROCESS_MASTER: 4
	  },
	  gPar: TRUE,
	  HardCodedPar: {
		DebounceOn : 2,
		DebounceOff : 2,
	  },
	  Operator: "TC_MON_OP_AND",
	  Logical: [
		`NOT gMain.Services.Recipes.Out.ParametersReady`
	  ]
	},
	MON_SYSTEM_HMI_STOP : {
	  Text: {
	      en: "HMI STOP Pressed",
	      es: "PARADA HMI Presionada",
	      fr: "ARRÊT IHM Appuyé",
	      de: "HMI-STOPP Gedrückt"
	    },
	  Sev: 4,
	  Mask: {
	      PROCESS_MASTER: 4
	  },
	  gPar: TRUE,
	  HardCodedPar: {
		DebounceOn : 2,
		DebounceOff : 2,
	  },
	  Operator: "TC_MON_OP_AND",
	  Logical: [
		`gIO.Safety.TC_IO_DI_HMI_STOP.Signal.Filtered`
	  ]
	}
}
```

- BuildVersion.ps1 - Pre-build script (not shown)

### Global.var - Global variables
```iecst
VAR
	gSim : Sim_typ;
	gIO : IO_typ;
	gVis : Vis_typ;
	gMain : Main_typ;
	gAlarmAddData : TC_AlarmX_AlarmExtraData_typ;
	gES : gES_typ;
	gScripts : Scripts_typ;
	JSONStrings : ARRAY[0..MAX_TC_SEQ_BUFFER_IDX] OF STRING[MAX_TC_SEQ_JSON_STRING_LEN];
	gDriver : Driver_typ;
END_VAR

VAR RETAIN
	gRemOK : BOOL;
	gPar : Par_typ;
	gRem : Rem_typ;
END_VAR
```

### Const.var - Global variables
```iecst
VAR CONSTANT
	STEPDELAY : DINT := 2;
	MAX_NOTIFICATION_IDX : DINT := 9; (*vis notification bar*)
	MAX_SEVERITY_IDX : DINT := 4;
	MAX_TC_RECIPE_IDX : DINT := 1;
	MAX_MON_IDX : DINT := 49;
	MAX_PROCESS_IDX : DINT := 2;
	MAX_MASTER_EVAL_IDX : DINT := 49;
	MAX_AXIS_R_IDX : DINT := 6;
	MAX_AXIS_V_IDX : DINT := 4;
	MAX_AXIS_A_IDX : DINT := MAX_AXIS_V_IDX+MAX_AXIS_R_IDX+1;
	MAX_VFD_IDX : DINT := 1;
	MAX_VFD_DATA_READ_IDX : DINT := 2;
	MAX_VFD_DATA_WRITE_IDX : DINT := 1;
END_VAR
(*Driver Constants*)
VAR CONSTANT
	MAX_DRIVER_FI_IDX : DINT := 0;
	MAX_DRIVER_FI_CMD_IDX : DINT := 13;
	MAX_DRIVER_FI_WAIT_IDX : DINT := 18;
	MAX_DRIVER_IN_IDX : DINT := 0;
	MAX_DRIVER_IN_CMD_IDX : DINT := 20;
	MAX_DRIVER_IN_WAIT_IDX : DINT := 18;
	MAX_DRIVER_IN_MON_IDX : DINT := 1;
	MAX_DRIVER_OU_IDX : DINT := 0;
	MAX_DRIVER_OU_CMD_IDX : DINT := 20;
	MAX_DRIVER_OU_WAIT_IDX : DINT := 18;
	MAX_DRIVER_OU_MON_IDX : DINT := 1;
	MAX_DRIVER_AB_IDX : DINT := MAX_AXIS_A_IDX;
	MAX_DRIVER_AB_CMD_IDX : DINT := 21;
	MAX_DRIVER_AB_WAIT_IDX : DINT := 18;
	MAX_DRIVER_AB_MON_IDX : DINT := 1;
	MAX_DRIVER_BX_IDX : DINT := 0;
	MAX_DRIVER_BX_CMD_IDX : DINT := 21;
	MAX_DRIVER_BX_WAIT_IDX : DINT := 18;
	MAX_DRIVER_BX_MON_IDX : DINT := 1;
	MAX_DRIVER_CS_IDX : DINT := MAX_AXIS_A_IDX;
	MAX_DRIVER_CS_CMD_IDX : DINT := 13;
	MAX_DRIVER_CS_WAIT_IDX : DINT := 12;
	MAX_DRIVER_CS_MON_IDX : DINT := 6;
	MAX_DRIVER_CS_SOURCE_IDX : DINT := 0;
	MAX_DRIVER_CN_IDX : DINT := 0;
	MAX_DRIVER_CN_CMD_IDX : DINT := 21;
	MAX_DRIVER_CN_WAIT_IDX : DINT := 18;
	MAX_DRIVER_CN_MON_IDX : DINT := 2;
	MAX_DRIVER_CN_SOURCE_IDX : DINT := 1;
	MAX_DRIVER_TR_IDX : DINT := 0;
	MAX_DRIVER_TR_CMD_IDX : DINT := 10;
	MAX_DRIVER_TR_WAIT_IDX : DINT := 0;
	MAX_DRIVER_TR_MON_IDX : DINT := 0;
	MAX_DRIVER_MR_IDX : DINT := 0;
	MAX_DRIVER_MR_CMD_IDX : DINT := 12;
	MAX_DRIVER_MR_WAIT_IDX : DINT := 4;
	MAX_DRIVER_MR_MON_IDX : DINT := 0;
END_VAR
```

### Enums.typ - Global data types
```iecst
TYPE
	DIR_MAN_ACTION_ENUM :
		( (*ENUM_STRING*)
		DIR_MAN_ACTION_NONE,
		DIR_MAN_ACTION_COPY_TO_USER,
		DIR_MAN_ACTION_COPY_TO_USB,
		DIR_MAN_ACTION_DELETE_USER,
		DIR_MAN_ACTION_DELETE_USB,
		DIR_MAN_ACTION_CREATE_DIR_USER,
		DIR_MAN_ACTION_CREATE_DIR_USB
		);
	DIR_MAN_STATE_ENUM :
		( (*ENUM_STRING*)
		DIR_MAN_RESET,
		DIR_MAN_DIRMAKE_CMD,
		DIR_MAN_DIRMAKE_WAIT,
		DIR_MAN_DIRREAD_CMD,
		DIR_MAN_DIRREAD_WAIT,
		DIR_MAN_DIRREAD_USB_CMD,
		DIR_MAN_DIRREAD_USB_WAIT,
		DIR_MAN_DIRSANITIZE_CMD,
		DIR_MAN_DIRSANITIZE_WAIT,
		DIR_MAN_TRANSFER_CMD,
		DIR_MAN_TRANSFER_WAIT,
		DIR_MAN_DELAY
		);
	TIME_STATE_ENUM :
		( (*ENUM_STRING*)
		TIME_RESET_C,
		TIME_CHECKPARREADY_W,
		TIME_IDLE_I,
		TIME_SET_C,
		TIME_SET_W,
		TIME_ERROR
		);
	RECIPE_ID_ENUM :
		( (*ENUM_STRING*)
		RECIPE_ID_REM,
		RECIPE_ID_PAR
		);
	MON_ENUM :
		( (*ENUM_STRING*)
		MON_SYSTEM_PAR_NOT_READY,
		MON_SYSTEM_HMI_STOP,
		MON_SAFETY_ESTOP,
		MON_RECIPE_REM_LOST_REM,
		MON_RECIPE_LOAD_BAD_REM,
		MON_RECIPE_LOAD_GOOD_REM,
		MON_RECIPE_GEN_ERR_REM,
		MON_RECIPE_REM_LOST_PAR,
		MON_RECIPE_LOAD_BAD_PAR,
		MON_RECIPE_LOAD_GOOD_PAR,
		MON_RECIPE_GEN_ERR_PAR
		);
	PROCESS_ENUM :
		( (*ENUM_STRING*)
		PROCESS_MASTER,
		PROCESS_TEMP
		);
	MASTER_EVAL_ENUM :
		( (*ENUM_STRING*)
		MASTER_EVAL_RESET,
		MASTER_EVAL_INIT,
		MASTER_EVAL_STOP_UNCONTROLLED,
		MASTER_EVAL_STOP_CONTROLLED,
		MASTER_EVAL_STOP_NORMAL,
		MASTER_EVAL_UNPAUSE,
		MASTER_EVAL_PAUSE,
		MASTER_EVAL_WAIT_BUFFER_EMPTY,
		MASTER_EVAL_START
		);
	MASTER_CALL_ENUM :
		( (*ENUM_STRING*)
		MASTER_CALL_IDLE,
		MASTER_CALL_RESET,
		MASTER_CALL_STOP_UNCONTROLLED,
		MASTER_CALL_STOP_CONTROLLED,
		MASTER_CALL_STOP_NORMAL,
		MASTER_CALL_UNPAUSE,
		MASTER_CALL_PAUSE,
		MASTER_CALL_START
		);
	DRIVER_INST_IN_ENUM :
		( (*ENUM_STRING*)
		DRIVER_INST_IN_0
		);
	C_IN_ENUM :
		( (*ENUM_STRING*)
		C_IN_RESET,
		C_IN_CLEARCMD,
		C_IN_CLEARMON,
		C_IN_DEFAULTMON,
		C_IN_CLEARPAR,
		C_IN_DEFAULTPAR,
		C_IN_SAVEPAR,
		C_IN_FORCEENABLE,
		C_IN_FORCEDISABLE
		);
	M_IN_ENUM :
		( (*ENUM_STRING*)
		M_IN_DI_ESTOP
		);
	W_IN_ENUM :
		( (*ENUM_STRING*)
		W_IN_DI_ESTOP
		);
	DRIVER_INST_DO_ENUM :
		( (*ENUM_STRING*)
		DRIVER_INST_DO_0
		);
	C_DO_ENUM :
		( (*ENUM_STRING*)
		C_DO_RESET,
		C_DO_CLEARCMD,
		C_DO_CLEARMON,
		C_DO_CLEARPAR,
		C_DO_DEFAULTMON,
		C_DO_DEFAULTPAR,
		C_DO_SAVEPAR,
		C_DO_ERRORRESET,
		C_DO_DISABLEALL,
		C_DO_ENABLE
		);
	M_DO_ENUM :
		( (*ENUM_STRING*)
		M_DO_ERROR
		);
	W_DO_ENUM :
		( (*ENUM_STRING*)
		W_DO_NOERROR
		);
	DRIVER_INST_AB_ENUM :
		( (*ENUM_STRING*)
		DRIVER_INST_AB_VX_0,
		DRIVER_INST_AB_VY_0,
		DRIVER_INST_AB_VZ_0,
		DRIVER_INST_AB_VT_0,
		DRIVER_INST_AB_VV_0,
		DRIVER_INST_AB_RX_0_0,
		DRIVER_INST_AB_RY_0_0,
		DRIVER_INST_AB_RZ_0_0,
		DRIVER_INST_AB_RT_0_0,
		DRIVER_INST_AB_RV_0_0,
		DRIVER_INST_AB_RP_0_0,
		DRIVER_INST_AB_RP_1_0
		);
	C_AB_ENUM :
		( (*ENUM_STRING*)
		C_AB_RESET,
		C_AB_CLEARCMD,
		C_AB_CLEARMON,
		C_AB_DEFAULTMON,
		C_AB_CLEARPAR,
		C_AB_DEFAULTPAR,
		C_AB_SAVEPAR,
		C_AB_LOADPAR,
		C_AB_ERRORRESET,
		C_AB_HOME,
		C_AB_POWER,
		C_AB_UPDATE,
		C_AB_AUTOTUNE,
		C_AB_JOGPOSITIVE,
		C_AB_JOGNEGATIVE,
		C_AB_LIMITLOAD,
		C_AB_STOP,
		C_AB_MOVEABSOLUTE,
		C_AB_MOVEADDITIVE,
		C_AB_MOVEVELOCITY,
		C_AB_RELEASEBRAKE,
		C_AB_SIMULATE
		);
	M_AB_ENUM :
		( (*ENUM_STRING*)
		M_AB_ERROR,
		M_AB_NOTPOWERON
		);
	W_AB_ENUM :
		( (*ENUM_STRING*)
		W_AB_NOERROR,
		W_AB_COMMUNICATIONREADY,
		W_AB_READYTOPOWERON,
		W_AB_POWERON,
		W_AB_ISHOMED,
		W_AB_LIMITLOADACTIVE,
		W_AB_MOVEDONE,
		W_AB_UPDATEDONE,
		W_AB_AUTOTUNEDONE,
		W_AB_BRAKERELEASED,
		W_AB_COMMANDABORTED,
		W_AB_COMMANDBUSY,
		W_AB_INPOSITION,
		W_AB_INVELOCITY,
		W_AB_MOVEACTIVE,
		W_AB_STOPPED,
		W_AB_JOGGING,
		W_AB_JOGLIMITREACHED,
		W_AB_SIMULATION
		);
	DRIVER_INST_CS_ENUM :
		( (*ENUM_STRING*)
		DRIVER_INST_CS_VX_0,
		DRIVER_INST_CS_VY_0,
		DRIVER_INST_CS_VZ_0,
		DRIVER_INST_CS_VT_0,
		DRIVER_INST_CS_VV_0,
		DRIVER_INST_CS_RX_0_0,
		DRIVER_INST_CS_RY_0_0,
		DRIVER_INST_CS_RZ_0_0,
		DRIVER_INST_CS_RT_0_0,
		DRIVER_INST_CS_RV_0_0
		);
	C_CS_ENUM :
		( (*ENUM_STRING*)
		C_CS_RESET,
		C_CS_CLEARCMD,
		C_CS_CLEARMON,
		C_CS_DEFAULTMON,
		C_CS_CLEARPAR,
		C_CS_DEFAULTPAR,
		C_CS_SAVEPAR,
		C_CS_LOADPAR,
		C_CS_ERRORRESET,
		C_CS_MOVECYCLICPOSITION,
		C_CS_MOVECYCLICVELOCITY,
		C_CS_TORQUECONTROL,
		C_CS_TORQUEFEEDFORWARD,
		C_CS_UPDATE
		);
	M_CS_ENUM :
		( (*ENUM_STRING*)
		M_CS_ERROR,
		M_CS_NOTMOVECYCLICPOSITIONACTIVE,
		M_CS_NOTMOVECYCLICVELOCITYACTIVE,
		M_CS_NOTTORQUECONTROLACTIVE,
		M_CS_NOTTORQUEFEEDFORWARDACTIVE,
		M_CS_TCAXISLIMITACTIVE,
		M_CS_NOTTCINTORQUE
		);
	W_CS_ENUM :
		( (*ENUM_STRING*)
		W_CS_NOERROR,
		W_CS_COMMANDABORTED,
		W_CS_COMMANDBUSY,
		W_CS_UPDATEDONE,
		W_CS_MOVECYCLICPOSITIONACTIVE,
		W_CS_MOVECYCLICVELOCITYACTIVE,
		W_CS_TORQUECONTROLACTIVE,
		W_CS_TORQUEFEEDFORWARDACTIVE,
		W_CS_TCAXISLIMITACTIVE,
		W_CS_TCDATAINITIALIZED,
		W_CS_TCINTORQUE,
		W_CS_TCREADY,
		W_CS_AXISREADY
		);
	DRIVER_INST_CN_ENUM :
		( (*ENUM_STRING*)
		DRIVER_INST_CN_0
		);
	C_CN_ENUM :
		( (*ENUM_STRING*)
		C_CN_RESET,
		C_CN_CLEARCMD,
		C_CN_CLEARMON,
		C_CN_DEFAULTMON,
		C_CN_CLEARPAR,
		C_CN_DEFAULTPAR,
		C_CN_SAVEPAR,
		C_CN_LOADPAR,
		C_CN_ERRORRESET,
		C_CN_HOME,
		C_CN_POWER,
		C_CN_UPDATE,
		C_CN_MOVEPROGRAM,
		C_CN_INTERRUPT,
		C_CN_CONTINUE,
		C_CN_STOP,
		C_CN_JOG,
		C_CN_MOVEBLOCK,
		C_CN_SINGLESTEP
		);
	M_CN_ENUM :
		( (*ENUM_STRING*)
		M_CN_ERROR,
		M_CN_NOTPOWERON,
		M_CN_NOTMOVEACTIVE
		);
	W_CN_ENUM :
		( (*ENUM_STRING*)
		W_CN_NOERROR,
		W_CN_COMMUNICATIONREADY,
		W_CN_READYTOPOWERON,
		W_CN_POWERON,
		W_CN_ISHOMED,
		W_CN_WAITFORCONTINUE,
		W_CN_MOVEDONE,
		W_CN_UPDATEDONE,
		W_CN_MOVEINTERRUPTED,
		W_CN_COMMANDABORTED,
		W_CN_COMMANDBUSY,
		W_CN_INMOTION,
		W_CN_MOVEACTIVE,
		W_CN_STOPPED,
		W_CN_SINGLESTEPACTIVE
		);
	DRIVER_INST_TR_ENUM :
		( (*ENUM_STRING*)
		DRIVER_INST_TR_0
		);
	C_TR_ENUM :
		( (*ENUM_STRING*)
		C_TR_RESET,
		C_TR_CLEARCMD,
		C_TR_CLEARMON,
		C_TR_DEFAULTMON,
		C_TR_CLEARPAR,
		C_TR_DEFAULTPAR,
		C_TR_SAVEPAR,
		C_TR_LOADPAR,
		C_TR_ERRORRESET,
		C_TR_ENABLE,
		C_TR_RESYNC
		);
	M_TR_ENUM :
		( (*ENUM_STRING*)
		M_TR_ERROR
		);
	W_TR_ENUM :
		( (*ENUM_STRING*)
		W_TR_NOERROR
		);
	TR_CONTROL_MODE_ENUM :
		(
		TR_CONTROL_MODE_ROTATE,
		TR_CONTROL_MODE_COORD,
		TR_CONTROL_MODE_TRANS
		);
	DRIVER_INST_MR_ENUM :
		( (*ENUM_STRING*)
		DRIVER_INST_MR_0
		);
	C_MR_ENUM :
		( (*ENUM_STRING*)
		C_MR_RESET,
		C_MR_CLEARCMD,
		C_MR_CLEARMON,
		C_MR_DEFAULTMON,
		C_MR_CLEARPAR,
		C_MR_DEFAULTPAR,
		C_MR_SAVEPAR,
		C_MR_LOADPAR,
		C_MR_ERRORRESET,
		C_MR_MBMOPEN,
		C_MR_MBMASTER,
		C_MR_MBMCLOSE,
		C_MR_MBMCMD
		);
	M_MR_ENUM :
		( (*ENUM_STRING*)
		M_MR_ERROR
		);
	W_MR_ENUM :
		( (*ENUM_STRING*)
		W_MR_NOERROR,
		W_MR_MBMOPEN,
		W_MR_MBMASTER,
		W_MR_MBMCLOSE,
		W_MR_MBMCMD
		);
	DRIVER_INST_BX_ENUM :
		( (*ENUM_STRING*)
		DRIVER_INST_BX_0
		);
	C_BX_ENUM :
		( (*ENUM_STRING*)
		C_BX_RESET,
		C_BX_CLEARCMD,
		C_BX_CLEARMON,
		C_BX_DEFAULTMON,
		C_BX_CLEARPAR,
		C_BX_DEFAULTPAR,
		C_BX_SAVEPAR,
		C_BX_LOADPAR,
		C_BX_ERRORRESET,
		C_BX_ENABLE
		);
	M_BX_ENUM :
		( (*ENUM_STRING*)
		M_BX_ERROR
		);
	W_BX_ENUM :
		( (*ENUM_STRING*)
		W_BX_NOERROR,
		W_BX_ACTIVE
		);
END_TYPE
```

### Rem.typ - Global data types
```iecst
TYPE
	Rem_typ : 	STRUCT
		UID : UDINT;
		RuntimeHours : REAL;
	END_STRUCT;
END_TYPE
```

### Services.typ - Global data types
```iecst
TYPE
	Services_typ : 	STRUCT
		DeviceName : STRING[255];
		Alarms : S_Alarms_typ;
		Recipes : S_Recipes_typ;
		DirMan : S_DirMan_typ;
		Time : S_Time_typ;
	END_STRUCT;
	S_Out_Status_typ : 	STRUCT
		CurrentState : STRING[80];
		InReset : BOOL;
		Initializing : BOOL;
		WaitingForCommand : BOOL;
		Processing : BOOL;
		InError : BOOL;
		Error : BOOL;
	END_STRUCT;
	S_Out_Ignore_typ : 	STRUCT
		Cmd : STRING[255];
		Reason : STRING[255];
	END_STRUCT;
	S_Out_ErrorInfo_typ : 	STRUCT
		Severity : USINT;
		Text : STRING[255];
		State : STRING[80];
		Code : UINT;
	END_STRUCT;
	S_Alarms_typ : 	STRUCT
		In : S_Alarms_In_typ;
		Internal : S_Alarms_Internal_typ;
		Out : S_Alarms_Out_typ;
	END_STRUCT;
	S_Alarms_In_typ : 	STRUCT
		ResetAlarms : BOOL;
		ClearHistory : BOOL;
		ExportHistory : BOOL;
		AlarmList : ARRAY[0..TC_ALARMX_BUFFER_IDX]OF TC_AlarmX_Core_Buffer_typ;
	END_STRUCT;
	S_Alarms_Internal_typ : 	STRUCT
		MpAlarmXListUI_0 : MpAlarmXListUI;
		MpAlarmXHistory_0 : MpAlarmXHistory;
		MpAlarmXCore_0 : MpAlarmXCore;
		CTON_StartDelay : CTON;
		CTON_ResetDelay : CTON;
		StateResetAlarms : INT;
		StateExportHistory : INT;
		MpAlarmXHistoryUI_0 : MpAlarmXHistoryUI;
		TC_AlarmXCore_0 : TC_AlarmXCore;
	END_STRUCT;
	S_Alarms_Out_typ : 	STRUCT
		AlarmActive : BOOL;
		BufferInfo : TC_AlarmX_BufferInfo_typ;
	END_STRUCT;
	S_Recipes_typ : 	STRUCT
		In : S_Recipes_In_typ;
		Internal : S_Recipes_Internal_typ;
		Out : S_Recipes_Out_typ;
	END_STRUCT;
	S_Recipes_In_typ : 	STRUCT
		ForceDefaults : BOOL;
		ForceSave : BOOL;
		ForceLoad : BOOL;
		RecipeDefinitions : ARRAY[0..MAX_TC_RECIPE_IDX]OF Recipe_Definition_typ;
	END_STRUCT;
	S_Recipes_Internal_typ : 	STRUCT
		TC_Recipe_Helper_0 : ARRAY[0..MAX_TC_RECIPE_IDX]OF TC_Recipe_Helper;
		tempAlarm : TC_AlarmX_Core_Buffer_typ;
	END_STRUCT;
	S_Recipes_Out_typ : 	STRUCT
		ParametersReady : BOOL;
	END_STRUCT;
	S_DirMan_typ : 	STRUCT
		In : S_DirMan_In_typ;
		Out : S_DirMan_Out_typ;
		Internal : S_DirMan_Internal_typ;
	END_STRUCT;
	S_DirMan_In_typ : 	STRUCT
		DirDef : ARRAY[0..MAX_DIR_DEF_IDX]OF TC_DirDef_typ;
		TransferList : ARRAY[0..MAX_TRANSFER_LIST_IDX]OF TC_Dir_Transfer_List_typ;
		Refresh : BOOL;
		RefreshDelay : LREAL;
	END_STRUCT;
	S_DirMan_Internal_typ : 	STRUCT
		State : DIR_MAN_STATE_ENUM;
		TC_DirReadAll_USB : TC_DirReadAll;
		TC_DirReadAll_0 : TC_DirReadAll;
		TC_DirSanitize_0 : TC_DirSanitize;
		TC_DirMake_0 : TC_DirMake;
		TC_Dir_USB_Connect_0 : TC_Dir_USB_Connect;
		TC_Dir_Transfer_0 : TC_Dir_Transfer;
		CTON_Delay : CTON;
	END_STRUCT;
	S_DirMan_Out_typ : 	STRUCT
		FileList : ARRAY[0..MAX_DIR_MAN_FILE_LIST_IDX]OF TC_FileList_typ;
		FileListUSB : ARRAY[0..MAX_DIR_MAN_FILE_LIST_IDX]OF TC_FileList_typ;
		DirectoriesCreated : BOOL;
	END_STRUCT;
	S_Time_typ : 	STRUCT
		In : S_Time_In_typ;
		Internal : S_Time_Internal_typ;
		Out : S_Time_Out_typ;
	END_STRUCT;
	S_Time_In_typ : 	STRUCT
		Cmd : S_Time_In_Cmd_typ;
		Par : S_Time_In_Par_typ;
	END_STRUCT;
	S_Time_In_Cmd_typ : 	STRUCT
		setTime : BOOL;
	END_STRUCT;
	S_Time_In_Par_typ : 	STRUCT
		newTime : DATE_AND_TIME;
	END_STRUCT;
	S_Time_Internal_typ : 	STRUCT
		state : TIME_STATE_ENUM;
		lastState : TIME_STATE_ENUM;
		CTON_Delay : CTON;
		CTON_Timeout : CTON;
		BlankCmdCmp : S_Time_In_Cmd_typ;
		DTSetTime_0 : DTSetTime;
		DTGetTime_0 : DTGetTime;
		tempAlarm : TC_AlarmX_Core_Buffer_typ;
		LastErrorInfo : S_Out_ErrorInfo_typ;
	END_STRUCT;
	S_Time_Out_typ : 	STRUCT
		Status : S_Time_Out_Status_typ;
		ErrorInfo : S_Out_ErrorInfo_typ;
		IgnoreInfo : S_Out_Ignore_typ;
	END_STRUCT;
	S_Time_Out_Status_typ : 	STRUCT
		CurrentState : STRING[80];
		InReset : BOOL;
		Initializing : BOOL;
		WaitingForCommand : BOOL;
		Processing : BOOL;
		InError : BOOL;
		Error : BOOL;
		TimeValid : BOOL;
		CurrentTime : DATE_AND_TIME;
	END_STRUCT;
END_TYPE
```

### Process.typ - Global data types
```iecst
TYPE
	Process_typ : 	STRUCT
		Monitor : P_Monitor_typ;
		Master : P_Master_typ;
	END_STRUCT;
	P_Monitor_typ : 	STRUCT
		Out : P_Monitor_Out_typ;
		In : P_Monitor_In_typ;
		Internal : P_Monitor_Internal_typ;
	END_STRUCT;
	P_Monitor_Out_typ : 	STRUCT
		SevActiveAny : BOOL;
		SevActive : ARRAY[0..MAX_SEVERITY_IDX]OF BOOL;
		ProcessErrorSev : ARRAY[0..MAX_PROCESS_IDX]OF DINT;
	END_STRUCT;
	P_Monitor_In_typ : 	STRUCT
		New_Member : USINT;
	END_STRUCT;
	P_Monitor_Internal_typ : 	STRUCT
		tempAlarm : TC_AlarmX_Core_Buffer_typ;
		TC_Mon_0 : ARRAY[0..MAX_MON_IDX]OF TC_Mon;
		TempSTRING : STRING[80];
	END_STRUCT;
	P_Master_typ : 	STRUCT
		In : P_Master_In_typ;
		Internal : P_Master_Internal_typ;
		Out : P_Master_Out_typ;
	END_STRUCT;
	P_Master_In_typ : 	STRUCT
		Par : P_Master_In_Par_typ;
		Cmd : P_Master_In_Cmd_typ;
	END_STRUCT;
	P_Master_In_Par_typ : 	STRUCT
		SingleStepMode : BOOL;
	END_STRUCT;
	P_Master_In_Cmd_typ : 	STRUCT
		Reset : BOOL;
		Start : BOOL;
		UncontrolledStop : BOOL;
		ControlledStop : BOOL;
		NormalStop : BOOL;
		Pause : BOOL;
		Unpause : BOOL;
		SingleStep : BOOL;
	END_STRUCT;
	P_Master_Internal_typ : 	STRUCT
		CALL : MASTER_CALL_ENUM;
		TC_Eval_0 : ARRAY[0..MAX_MASTER_EVAL_IDX]OF TC_Eval;
		TC_Seq_Handler_0 : TC_Seq_Handler;
	END_STRUCT;
	P_Master_Out_IgnoreInfo_typ : 	STRUCT
		Cmd : STRING[255];
		Reason : STRING[255];
	END_STRUCT;
	P_Master_Out_ErrorInfo_typ : 	STRUCT
		Severity : DINT;
		Text : STRING[255];
	END_STRUCT;
	P_Master_Out_Status_typ : 	STRUCT
		CurrentState : STRING[80];
		Stopping : BOOL;
		Paused : BOOL;
		InReset : BOOL;
		Initializing : BOOL;
		WaitingForCommand : BOOL;
		SingleStepWaiting : BOOL;
		Processing : BOOL;
		InError : BOOL;
		Error : BOOL;
	END_STRUCT;
	P_Master_Out_typ : 	STRUCT
		IgnoreInfo : P_Master_Out_IgnoreInfo_typ;
		ErrorInfo : P_Master_Out_ErrorInfo_typ;
		Status : P_Master_Out_Status_typ;
	END_STRUCT;
END_TYPE
```

### IO.typ - Global data types
```iecst
TYPE
	IO_typ : 	STRUCT
		ForceEnable : BOOL;
		AllConfiguredModulesOk : BOOL;
		Safety : IO_Safety_typ;
		BX18 : IO_BX18_typ;
		VFD : ARRAY[0..MAX_VFD_IDX]OF IO_VFD_typ;
		Motion : IO_Motion_typ;
	END_STRUCT;
	IO_Safety_typ : 	STRUCT
		TC_IO_DI_HMI_STOP : TC_IO_DI;
		TC_IO_DI_ESTOP : TC_IO_DI;
	END_STRUCT;
	IO_BX18_typ : 	STRUCT
		TC_IO_DI_ReqSettingsInvalid : TC_IO_DI;
		TC_IO_DI_ReqStateInvalid : TC_IO_DI;
		TC_IO_DI_EDMOutputActive : TC_IO_DI;
		TC_IO_DI_EdgefindModeEnabled : TC_IO_DI;
		TC_IO_DI_EdgeFound : TC_IO_DI;
		TC_IO_DI_ISOPulseMode : TC_IO_DI;
		TC_IO_DI_ElectrodePositiveMode : TC_IO_DI;
		TC_IO_DI_PowerFault : TC_IO_DI;
		TC_IO_DI_LowVoltageFault : TC_IO_DI;
		TC_IO_DI_HighVoltageFault : TC_IO_DI;
		TC_IO_DI_EstopActive : TC_IO_DI;
		TC_IO_DI_OnTimeChanged : TC_IO_DI;
		TC_IO_DI_OffTimeChanged : TC_IO_DI;
		TC_IO_DI_CurrentChanged : TC_IO_DI;
		TC_IO_AI_Feedback : TC_IO_AI;
		TC_IO_AI_Power : TC_IO_AI;
		TC_IO_DO_Enable : TC_IO_DO;
		TC_IO_DO_ISOFreqMode : TC_IO_DO;
		TC_IO_DO_EdgeFindMode : TC_IO_DO;
		TC_IO_DO_ElectrodePositiveMode : TC_IO_DO;
		TC_IO_DO_ChangeRequest : TC_IO_DO;
		TC_IO_AO_OnTime : TC_IO_AO;
		TC_IO_AO_OffTime : TC_IO_AO;
		TC_IO_AO_Current : TC_IO_AO;
		ModuleOK : BOOL;
		Outputs_control : UINT;
		Outputs_onTime : UINT;
		Outputs_offTime : UINT;
		Outputs_current : UINT;
		Inputs_status : UINT;
		Inputs_EDMservofeedback : UINT;
		Inputs_power : UINT;
	END_STRUCT;
	IO_VFD_typ : 	STRUCT
		EventWrite : ARRAY[0..MAX_VFD_DATA_WRITE_IDX]OF BOOL;
		DataWrite : ARRAY[0..MAX_VFD_DATA_WRITE_IDX]OF UINT;
		DataWriteCmp : ARRAY[0..MAX_VFD_DATA_WRITE_IDX]OF UINT;
		EventRead : ARRAY[0..MAX_VFD_DATA_READ_IDX]OF BOOL;
		DataRead : ARRAY[0..MAX_VFD_DATA_READ_IDX]OF UINT;
		CTON_AutoWrite : CTON;
		RFRD : INT;
		LFRD : INT;
		LFT : UINT;
		CMD : UINT;
		ETA : UINT;
	END_STRUCT;
	IO_Motion_typ : 	STRUCT
		ModuleOK : BOOL;
		ENABLE : BOOL;
		ENABLED : BOOL;
		StepDelay : DINT := 2;
		SetPosition : DINT;
		ActualPosition : DINT;
		Home : DINT;
		SwitchOn : BOOL;
		SwitchedOn : BOOL;
		TC_IO_DI_HomeSwitchZ : TC_IO_DI;
	END_STRUCT;
END_TYPE
```

### Sim.typ - Global data types
```iecst
TYPE
	Sim_Time_typ : 	STRUCT
		RTInfo_0 : RTInfo;
		TimeInc : LREAL;
		Time : LREAL;
	END_STRUCT;
	Sim_typ : 	STRUCT
		Full : BOOL;
		IO : BOOL;
		Time : Sim_Time_typ;
	END_STRUCT;
END_TYPE
```

### Main.typ - Global data types
```iecst
TYPE
	Main_typ : 	STRUCT
		ErrorReset : BOOL;
		Process : Process_typ;
		Services : Services_typ;
	END_STRUCT;
	Scripts_typ : 	STRUCT
		FirstStart : ARRAY[0..MAX_TC_SEQ_BUFFER_IDX]OF STRING[MAX_TC_SEQ_JSON_STRING_LEN];
	END_STRUCT;
END_TYPE
```

### Driver.typ - Global data types
```iecst
TYPE
	Driver_typ : 	STRUCT
		ResetAll : BOOL;
		IN : ARRAY[0..MAX_DRIVER_IN_IDX]OF Driver_IN_typ;
		BX : ARRAY[0..MAX_DRIVER_BX_IDX]OF Driver_BX_typ;
		AB : ARRAY[0..MAX_DRIVER_AB_IDX]OF Driver_AB_typ;
		CS : ARRAY[0..MAX_DRIVER_CS_IDX]OF Driver_CS_typ;
		CN : ARRAY[0..MAX_DRIVER_CN_IDX]OF Driver_CN_typ;
		TR : ARRAY[0..MAX_DRIVER_TR_IDX]OF Driver_TR_typ;
		MR : ARRAY[0..MAX_DRIVER_MR_IDX]OF Driver_MR_typ;
		FI : ARRAY[0..MAX_DRIVER_FI_IDX]OF Driver_FI_typ;
		OU : ARRAY[0..MAX_DRIVER_OU_IDX]OF Driver_OU_typ;
	END_STRUCT;
	Driver_Par_Mon_typ : 	STRUCT
		Enable : BOOL;
		Sev : DINT;
		Time : LREAL;
	END_STRUCT;
	Driver_CS_typ : 	STRUCT
		Cmd : ARRAY[0..MAX_DRIVER_CS_CMD_IDX]OF BOOL;
		Wait : ARRAY[0..MAX_DRIVER_CS_WAIT_IDX]OF DINT;
		Mon : ARRAY[0..MAX_DRIVER_CS_MON_IDX]OF BOOL;
		Sev : ARRAY[0..MAX_DRIVER_CS_MON_IDX]OF DINT;
		CTON_Mon : ARRAY[0..MAX_DRIVER_CS_MON_IDX]OF CTON;
		DefaultPar : Driver_CS_Par_typ;
		Par : Driver_CS_Par_typ;
		Status : Driver_CS_Status_typ;
		MpAxisCyclicSet_0 : MpAxisCyclicSet;
		MpLinkADR : UDINT;
		CyclicPositionSetpoint : ARRAY[0..MAX_DRIVER_CS_SOURCE_IDX]OF LREAL;
		CyclicTorqueSetpoint : ARRAY[0..MAX_DRIVER_CS_SOURCE_IDX]OF REAL;
		CyclicTorqueFeedForwardSetpoint : ARRAY[0..MAX_DRIVER_CS_SOURCE_IDX]OF REAL;
		CyclicVelocitySetpoint : ARRAY[0..MAX_DRIVER_CS_SOURCE_IDX]OF REAL;
		FirstScanComplete : BOOL;
		ParametersLoaded : BOOL;
	END_STRUCT;
	Driver_CS_Par_typ : 	STRUCT
		Mon : ARRAY[0..MAX_DRIVER_CS_MON_IDX]OF Driver_Par_Mon_typ;
		CS : MpAxisCyclicSetParType;
		CyclicPositionSource : DINT;
		CyclicTorqueSource : DINT;
		CyclicTorqueFeedForwardSource : DINT;
		CyclicVelocitySource : DINT;
	END_STRUCT;
	Driver_CS_Status_typ : 	STRUCT
		Severity : DINT;
	END_STRUCT;
	Driver_AB_typ : 	STRUCT
		Cmd : ARRAY[0..MAX_DRIVER_AB_CMD_IDX]OF BOOL;
		Wait : ARRAY[0..MAX_DRIVER_AB_WAIT_IDX]OF DINT;
		Mon : ARRAY[0..MAX_DRIVER_AB_MON_IDX]OF BOOL;
		Sev : ARRAY[0..MAX_DRIVER_AB_MON_IDX]OF DINT;
		CTON_Mon : ARRAY[0..MAX_DRIVER_AB_MON_IDX]OF CTON;
		Par : Driver_AB_Par_typ;
		DefaultPar : Driver_AB_Par_typ;
		Status : Driver_AB_Status_typ;
		MpAxisBasic_0 : MpAxisBasic;
		MpLinkADR : UDINT;
		FirstScanComplete : BOOL;
		ParametersLoaded : BOOL;
	END_STRUCT;
	Driver_AB_Par_typ : 	STRUCT
		Mon : ARRAY[0..MAX_DRIVER_AB_MON_IDX]OF Driver_Par_Mon_typ;
		AB : MpAxisBasicParType;
	END_STRUCT;
	Driver_AB_Status_typ : 	STRUCT
		Position : LREAL;
		Velocity : LREAL;
		Severity : DINT;
	END_STRUCT;
	Driver_FI_typ : 	STRUCT
		Cmd : ARRAY[0..MAX_DRIVER_FI_CMD_IDX]OF BOOL;
		Wait : ARRAY[0..MAX_DRIVER_FI_WAIT_IDX]OF DINT;
		Par : Driver_FI_Par_typ;
		FileClose : FileClose;
		FileCopy : FileCopy;
		FileCreate : FileCreate;
		FileDelete : FileDelete;
		FileInfo : FileInfo;
		FileOpen : FileOpen;
		FileReadEx : FileReadEx;
		FileRename : FileRename;
		FileTruncate : FileTruncate;
		FileWriteEx : FileWriteEx;
		DirCopy : DirCopy;
		DirCreate : DirCreate;
		DirDeleteEx : DirDeleteEx;
		DirInfo : DirInfo;
		DirOpen : DirOpen;
		DirReadEx : DirReadEx;
		DirRename : DirRename;
		DirClose : DirClose;
		GetAttributes : GetAttributes;
		SetAttributes : SetAttributes;
		GetVolumeLabel : GetVolumeLabel;
		GetVolumeSerialNo : GetVolumeSerialNo;
		DevLink : DevLink;
		DevMemInfo : DevMemInfo;
		DevUnlink : DevUnlink;
	END_STRUCT;
	Driver_FI_Par_typ : 	STRUCT
		FileName : STRING[255];
	END_STRUCT;
	Driver_CN_typ : 	STRUCT
		Cmd : ARRAY[0..MAX_DRIVER_CN_CMD_IDX]OF BOOL;
		Wait : ARRAY[0..MAX_DRIVER_CN_WAIT_IDX]OF DINT;
		Mon : ARRAY[0..MAX_DRIVER_CN_MON_IDX]OF BOOL;
		Sev : ARRAY[0..MAX_DRIVER_CN_MON_IDX]OF DINT;
		CTON_Mon : ARRAY[0..MAX_DRIVER_CN_MON_IDX]OF CTON;
		Par : Driver_CN_Par_typ;
		DefaultPar : Driver_CN_Par_typ;
		Status : Driver_CN_Status_typ;
		MpCncFlex_0 : MpCncFlex;
		MC_GroupReadActualPosition_15_0 : MC_GroupReadActualPosition_15;
		MpLinkADR : UDINT;
		OverrideSetpoint : ARRAY[0..MAX_DRIVER_CN_SOURCE_IDX]OF REAL;
		RapidOverrideSetpoint : ARRAY[0..MAX_DRIVER_CN_SOURCE_IDX]OF REAL;
		FeedrateOverrideSetpoint : ARRAY[0..MAX_DRIVER_CN_SOURCE_IDX]OF REAL;
		FirstScanComplete : BOOL;
		ParametersLoaded : BOOL;
	END_STRUCT;
	Driver_CN_Par_typ : 	STRUCT
		Mon : ARRAY[0..MAX_DRIVER_CN_MON_IDX]OF Driver_Par_Mon_typ;
		CN : MpCncFlexParType;
		OverrideSource : DINT;
		RapidOverrideSource : DINT;
		FeedrateOverrideSource : DINT;
		Kinematics : ARRAY[0..14]OF LREAL;
	END_STRUCT;
	Driver_CN_Status_typ : 	STRUCT
		Severity : DINT;
		Position : ARRAY[0..14]OF LREAL;
		Position_mcJACS : ARRAY[0..14]OF LREAL;
		PathVelocity : REAL;
		Info : MpCncFlexInfoType;
	END_STRUCT;
	Driver_IN_typ : 	STRUCT
		Cmd : ARRAY[0..MAX_DRIVER_IN_CMD_IDX]OF BOOL;
		Wait : ARRAY[0..MAX_DRIVER_IN_WAIT_IDX]OF DINT;
		Mon : ARRAY[0..MAX_DRIVER_IN_MON_IDX]OF BOOL;
		Sev : ARRAY[0..MAX_DRIVER_IN_MON_IDX]OF DINT;
		CTON_Mon : ARRAY[0..MAX_DRIVER_IN_MON_IDX]OF CTON;
		Par : Driver_IN_Par_typ;
		DefaultPar : Driver_IN_Par_typ;
		Status : Driver_IN_Status_typ;
		FirstScanComplete : BOOL;
		New_Member : USINT;
		DI_Estop : TC_IO_DI;
	END_STRUCT;
	Driver_IN_Par_typ : 	STRUCT
		Mon : ARRAY[0..MAX_DRIVER_IN_MON_IDX]OF Driver_Par_Mon_typ;
		ForceEnable : BOOL;
		DI_Estop_Par : TC_IO_Digital_Par_typ;
		DI_Estop_Forcing : TC_IO_Digital_Forcing_typ;
		DI_Estop_Sim : TC_IO_Digital_Sim_typ;
	END_STRUCT;
	Driver_IN_Status_typ : 	STRUCT
		Severity : DINT;
	END_STRUCT;
	Driver_OU_typ : 	STRUCT
		Cmd : ARRAY[0..MAX_DRIVER_OU_CMD_IDX]OF BOOL;
		Wait : ARRAY[0..MAX_DRIVER_OU_WAIT_IDX]OF DINT;
		Mon : ARRAY[0..MAX_DRIVER_OU_MON_IDX]OF BOOL;
		Sev : ARRAY[0..MAX_DRIVER_OU_MON_IDX]OF DINT;
		CTON_Mon : ARRAY[0..MAX_DRIVER_OU_MON_IDX]OF CTON;
		Par : Driver_OU_Par_typ;
		DefaultPar : Driver_OU_Par_typ;
		Status : Driver_OU_Status_typ;
		FirstScanComplete : BOOL;
		DO_Enable : TC_IO_DO;
	END_STRUCT;
	Driver_OU_Par_typ : 	STRUCT
		Mon : ARRAY[0..MAX_DRIVER_OU_MON_IDX]OF Driver_Par_Mon_typ;
		DO_Enable : TC_IO_Digital_Par_typ;
	END_STRUCT;
	Driver_OU_Status_typ : 	STRUCT
		Severity : DINT;
	END_STRUCT;
	Driver_TR_typ : 	STRUCT
		Cmd : ARRAY[0..MAX_DRIVER_TR_CMD_IDX]OF BOOL;
		Wait : ARRAY[0..MAX_DRIVER_TR_WAIT_IDX]OF DINT;
		Mon : ARRAY[0..MAX_DRIVER_TR_MON_IDX]OF BOOL;
		Sev : ARRAY[0..MAX_DRIVER_TR_MON_IDX]OF DINT;
		CTON_Mon : ARRAY[0..MAX_DRIVER_TR_MON_IDX]OF CTON;
		DefaultPar : Driver_TR_Par_typ;
		Par : Driver_TR_Par_typ;
		Status : Driver_TR_Status_typ;
		FirstScanComplete : BOOL;
		ParametersLoaded : BOOL;
	END_STRUCT;
	Driver_TR_Par_typ : 	STRUCT
		Mon : ARRAY[0..MAX_DRIVER_TR_MON_IDX]OF Driver_Par_Mon_typ;
		ControlMode : TR_CONTROL_MODE_ENUM;
		WorldCoordMode : BOOL;
		VelocityFactor : LREAL;
		Filter : LREAL;
		Gain : REAL;
		IntegralTime : REAL;
	END_STRUCT;
	Driver_TR_Status_typ : 	STRUCT
		Active : BOOL;
		Severity : DINT;
		TotalLag : LREAL;
		Lag : ARRAY[0..14]OF LREAL;
		SetTCP : ARRAY[0..14]OF LREAL;
		SetJoint : ARRAY[0..14]OF LREAL;
		TcpMatrix : ARRAY[0..3,0..3]OF LREAL;
		TcpSetpoint : ARRAY[0..14]OF LREAL;
		TcpSetpointLastStable : ARRAY[0..14]OF LREAL;
		InputCmd : ARRAY[0..14]OF LREAL;
		LimitedCmd : ARRAY[0..14]OF LREAL;
		VelCmd : ARRAY[0..14]OF LREAL;
		VelCmd_World : ARRAY[0..14]OF LREAL;
		Override : LREAL;
		MTBasicsPID_0 : ARRAY[0..14]OF MTBasicsPID;
	END_STRUCT;
	Driver_MR_typ : 	STRUCT
		Cmd : ARRAY[0..MAX_DRIVER_MR_CMD_IDX]OF BOOL;
		Wait : ARRAY[0..MAX_DRIVER_MR_WAIT_IDX]OF DINT;
		Mon : ARRAY[0..MAX_DRIVER_MR_MON_IDX]OF BOOL;
		Sev : ARRAY[0..MAX_DRIVER_MR_MON_IDX]OF DINT;
		CTON_Mon : ARRAY[0..MAX_DRIVER_MR_MON_IDX]OF CTON;
		DefaultPar : Driver_MR_Par_typ;
		Par : Driver_MR_Par_typ;
		Status : Driver_MR_Status_typ;
		FirstScanComplete : BOOL;
		ParametersLoaded : BOOL;
		Ident : UDINT;
		MBMOpen_0 : MBMOpen;
		MBMaster_0 : MBMaster;
		MBMCmd_0 : MBMCmd;
		MBMClose_0 : MBMClose;
	END_STRUCT;
	Driver_MR_Par_typ : 	STRUCT
		Mon : ARRAY[0..MAX_DRIVER_TR_MON_IDX]OF Driver_Par_Mon_typ;
		Device : STRING[255];
		Mode : STRING[255];
		DataObject : STRING[255];
		IsAscii : BOOL;
		Timeout : LREAL;
		CmdNode : UDINT;
		CmdFunctionCall : UDINT;
		CmdOffset : UDINT;
		CmdData : UINT;
	END_STRUCT;
	Driver_MR_Status_typ : 	STRUCT
		Active : BOOL;
		Severity : DINT;
	END_STRUCT;
	Driver_BX_typ : 	STRUCT
		Cmd : ARRAY[0..MAX_DRIVER_BX_CMD_IDX]OF BOOL;
		Wait : ARRAY[0..MAX_DRIVER_BX_WAIT_IDX]OF DINT;
		Mon : ARRAY[0..MAX_DRIVER_BX_MON_IDX]OF BOOL;
		Sev : ARRAY[0..MAX_DRIVER_BX_MON_IDX]OF DINT;
		CTON_Mon : ARRAY[0..MAX_DRIVER_BX_MON_IDX]OF CTON;
		Par : Driver_BX_Par_typ;
		DefaultPar : Driver_BX_Par_typ;
		Status : Driver_BX_Status_typ;
		FirstScanComplete : BOOL;
		ParametersLoaded : BOOL;
		MTBasicsPID_0 : MTBasicsPID;
	END_STRUCT;
	Driver_BX_Par_typ : 	STRUCT
		Mon : ARRAY[0..MAX_DRIVER_BX_MON_IDX]OF Driver_Par_Mon_typ;
		EdgeFindMode : BOOL;
		ISOPulseMode : BOOL;
		ElectrodePositiveMode : BOOL;
		PID : MTPIDParametersType;
		SetFeedback : REAL;
		MinOverrideFactor : REAL;
		MaxOverrideFactor : REAL;
		Current : REAL;
		OnTime : REAL;
		OffTime : REAL;
	END_STRUCT;
	Driver_BX_Status_typ : 	STRUCT
		Severity : DINT;
		OverrideFactor : REAL;
		SetOffTime : REAL;
		SetOnTime : REAL;
		SetCurrent : REAL;
		ActualPower : REAL;
		SetFeedback : REAL;
		ActualFeedback : REAL;
		OutputActive : BOOL;
		EdgeFindEnabled : BOOL;
		EdgeFound : BOOL;
		ISOPulseMode : BOOL;
		ElectrodePositiveMode : BOOL;
		StateInvalid : BOOL;
		SettingsInvalid : BOOL;
		PowerFault : BOOL;
		LowVoltageFault : BOOL;
		HighVoltageFault : BOOL;
		EstopActive : BOOL;
	END_STRUCT;
END_TYPE
```

### Par.typ - Global data types
```iecst
TYPE
	Par_typ : 	STRUCT
		IO : Par_IO_typ;
		System : Par_System_typ; (*Desc 1*) (*Desc 2*) (*Desc 3*)
		Process : Par_Process_typ;
		Services : Par_Services_typ;
		Driver : Par_Driver_typ;
	END_STRUCT;
	Par_Services_typ : 	STRUCT
		Cert : Par_Services_Cert_typ;
		Email : Par_Services_Email_typ;
	END_STRUCT;
	Par_Services_Cert_typ : 	STRUCT
		CountryCode : STRING[9];
		StateProvince : STRING[513];
		Locality : STRING[513];
		Organization : STRING[255];
		OrganizationUnit : STRING[255];
		ContactEmail : STRING[513];
		CommonName : STRING[255];
		IP : STRING[513];
	END_STRUCT;
	Par_Services_Email_typ : 	STRUCT
		Port : UINT;
		Timeout : UDINT;
		Host : STRING[255];
		User : STRING[255];
		Password : STRING[255];
		Sender : STRING[255];
		Receiver : STRING[255];
	END_STRUCT;
	Par_Process_typ : 	STRUCT
		Master : Par_Master_typ;
		Monitor : Par_Monitor_typ;
	END_STRUCT;
	Par_System_typ : 	STRUCT
		Debugger : Par_System_Debugger_typ;
		UnitCode : STRING[20];
		LanguageCode : STRING[20];
		Serial : STRING[80];
	END_STRUCT;
	Par_Monitor_typ : 	STRUCT
		Mon : ARRAY[0..MAX_MON_IDX]OF TC_Mon_Par_typ := [(FilterOnTime:=10.0,FilterOffTime:=5.0),49(0)];
	END_STRUCT;
	Par_Master_typ : 	STRUCT
		Eval : ARRAY[0..MAX_MASTER_EVAL_IDX]OF TC_Eval_Par_typ;
	END_STRUCT;
	Par_System_Debugger_typ : 	STRUCT
		HoldProcessInInit : BOOL;
	END_STRUCT;
	Par_IO_Motion_typ : 	STRUCT
		TC_IO_DI_HomeSwitchX : TC_IO_Digital_Par_typ;
		TC_IO_DI_HomeSwitchY : TC_IO_Digital_Par_typ;
		TC_IO_DI_HomeSwitchZ : TC_IO_Digital_Par_typ;
	END_STRUCT;
	Par_IO_BX18_typ : 	STRUCT
		TC_IO_DI_ReqSettingsInvalid : TC_IO_Digital_Par_typ;
		TC_IO_DI_ReqStateInvalid : TC_IO_Digital_Par_typ;
		TC_IO_DI_EDMOutputActive : TC_IO_Digital_Par_typ;
		TC_IO_DI_EdgefindModeEnabled : TC_IO_Digital_Par_typ;
		TC_IO_DI_EdgeFound : TC_IO_Digital_Par_typ;
		TC_IO_DI_ISOPulseMode : TC_IO_Digital_Par_typ;
		TC_IO_DI_ElectrodePositiveMode : TC_IO_Digital_Par_typ;
		TC_IO_DI_PowerFault : TC_IO_Digital_Par_typ;
		TC_IO_DI_LowVoltageFault : TC_IO_Digital_Par_typ;
		TC_IO_DI_HighVoltageFault : TC_IO_Digital_Par_typ;
		TC_IO_DI_EstopActive : TC_IO_Digital_Par_typ;
		TC_IO_DI_OnTimeChanged : TC_IO_Digital_Par_typ;
		TC_IO_DI_OffTimeChanged : TC_IO_Digital_Par_typ;
		TC_IO_DI_CurrentChanged : TC_IO_Digital_Par_typ;
		TC_IO_AI_Feedback : TC_IO_Analog_Par_typ;
		TC_IO_AI_Power : TC_IO_Analog_Par_typ;
		TC_IO_DO_Enable : TC_IO_Digital_Par_typ;
		TC_IO_DO_ISOFreqMode : TC_IO_Digital_Par_typ;
		TC_IO_DO_EdgeFindMode : TC_IO_Digital_Par_typ;
		TC_IO_DO_ElectrodePositiveMode : TC_IO_Digital_Par_typ;
		TC_IO_DO_ChangeRequest : TC_IO_Digital_Par_typ;
		TC_IO_AO_OnTime : TC_IO_Analog_Par_typ;
		TC_IO_AO_OffTime : TC_IO_Analog_Par_typ;
		TC_IO_AO_Current : TC_IO_Analog_Par_typ;
	END_STRUCT;
	Par_IO_Safety_typ : 	STRUCT
		TC_IO_DI_HMI_STOP : TC_IO_Digital_Par_typ;
		TC_IO_DI_ESTOP : TC_IO_Digital_Par_typ;
	END_STRUCT;
	Par_IO_typ : 	STRUCT
		Simulate : BOOL;
		Safety : Par_IO_Safety_typ;
		BX18 : Par_IO_BX18_typ;
		Motion : Par_IO_Motion_typ;
	END_STRUCT;
	Par_Driver_typ : 	STRUCT
		BX : ARRAY[0..MAX_DRIVER_BX_IDX]OF Driver_BX_Par_typ;
		AB : ARRAY[0..MAX_DRIVER_AB_IDX]OF Driver_AB_Par_typ;
		CS : ARRAY[0..MAX_DRIVER_CS_IDX]OF Driver_CS_Par_typ;
		CN : ARRAY[0..MAX_DRIVER_CN_IDX]OF Driver_CN_Par_typ;
		TR : ARRAY[0..MAX_DRIVER_TR_IDX]OF Driver_TR_Par_typ;
		MR : ARRAY[0..MAX_DRIVER_MR_IDX]OF Driver_MR_Par_typ;
	END_STRUCT;
END_TYPE
```

### Vis.typ - Global data types
```iecst
TYPE
	Vis_typ : 	STRUCT
		Navigation : Vis_Navigation_typ;
		Header : Vis_Header_typ;
		Footer : Vis_Footer_typ;
		Alarms : Vis_Alarms_typ;
		Settings : Vis_Settings_typ;
		Services : Vis_Services_typ;
	END_STRUCT;
	Vis_Navigation_typ : 	STRUCT
		STOP : BOOL;
	END_STRUCT;
	Vis_Footer_typ : 	STRUCT
		IdentifyConfig_0 : IdentifyConfig;
		Revision : STRING[300];
		Start : BOOL;
		Pause : BOOL;
		Stop : BOOL;
		SetTime : BOOL;
		currentTime : DATE_AND_TIME;
		newTime : DATE_AND_TIME;
		TimeNotValid : BOOL;
		CTON_Init : CTON;
	END_STRUCT;
	Vis_Header_typ : 	STRUCT
		Monitor : Vis_Header_Monitor_typ;
		Notifications : Vis_Header_Notifications_typ;
	END_STRUCT;
	Vis_Header_Notifications_typ : 	STRUCT
		Visible : ARRAY[0..MAX_NOTIFICATION_IDX]OF BOOL;
	END_STRUCT;
	Vis_Header_Monitor_typ : 	STRUCT
		Styles : Vis_Header_Monitor_Styles_typ;
	END_STRUCT;
	Vis_Header_Monitor_Styles_typ : 	STRUCT
		Text : STRING[8];
		Background : STRING[8];
		GridColor : STRING[8];
		Line0 : STRING[8];
		Line1 : STRING[8];
		Line2 : STRING[8];
		Line3 : STRING[8];
	END_STRUCT;
	Vis_Alarms_typ : 	STRUCT
		Active : Vis_Alarms_Active_typ;
		History : Vis_Alarms_History_typ;
	END_STRUCT;
	Vis_Alarms_Active_typ : 	STRUCT
		UIConnect : MpAlarmXListUIConnectType;
		Reset : BOOL;
		PageDown : BOOL;
		PageUp : BOOL;
		SelectedIndex : UINT;
		TableConfig : STRING[255];
		TempINT : INT;
		TempSTRING : STRING[30];
	END_STRUCT;
	Vis_Alarms_History_typ : 	STRUCT
		UIConnect : MpAlarmXHistoryUIConnectType;
		State : ARRAY[0..49]OF UINT;
		Clear : BOOL;
		PageDown : BOOL;
		PageUp : BOOL;
		Export : BOOL;
		SelectedIndex : UINT;
		TableConfig : STRING[255];
		TempINT : INT;
		TempSTRING : STRING[30];
	END_STRUCT;
	Vis_Settings_Save_typ : 	STRUCT
		Modified : BOOL;
		Save : BOOL;
		Cancel : BOOL;
	END_STRUCT;
	Vis_Settings_typ : 	STRUCT
		Par : Par_typ;
		ParCmp : Par_typ;
		Save : Vis_Settings_Save_typ;
	END_STRUCT;
	Vis_Services_typ : 	STRUCT
		DirMan : Vis_Services_DirMan_typ;
	END_STRUCT;
	Vis_Services_DirMan_typ : 	STRUCT
		FileList : Vis_Services_DirMan_FileList_typ;
		FileListUSB : Vis_Services_DirMan_FileList_typ;
		DirectoriesCreated : BOOL;
		UpdatingEdge : BOOL;
		Updating : BOOL;
		Refresh : BOOL;
		Cancel : BOOL;
		Confirm : BOOL;
		Command : BOOL;
		USBConnected : BOOL;
		CmdInactive : BOOL;
		CmdActive : BOOL;
		ActiveCmd : Vis_Services_DirMan_Cmd_typ;
		Cmd : Vis_Services_DirMan_Cmd_typ;
		Enable_Command : BOOL;
		Busy : BOOL;
		SelectedIndexUser : INT;
		SelectedIndexUSB : INT;
		TempSTRING : STRING[80];
		TempINT : INT;
		TableConfig_USB : STRING[255];
		TableConfig_User : STRING[255];
	END_STRUCT;
	Vis_Services_DirMan_FileList_typ : 	STRUCT
		Num : ARRAY[0..MAX_DIR_MAN_FILE_LIST_IDX]OF UDINT;
		Path : ARRAY[0..MAX_DIR_MAN_FILE_LIST_IDX]OF STRING[260];
		DateString : ARRAY[0..MAX_DIR_MAN_FILE_LIST_IDX]OF STRING[25];
		Size : ARRAY[0..MAX_DIR_MAN_FILE_LIST_IDX]OF UDINT;
		IsDir : ARRAY[0..MAX_DIR_MAN_FILE_LIST_IDX]OF BOOL;
	END_STRUCT;
	Vis_Services_DirMan_Cmd_typ : 	STRUCT
		Action : DIR_MAN_ACTION_ENUM;
		DirUSB : BOOL;
		DirUser : BOOL;
		PathUSB : STRING[260];
		PathUser : STRING[260];
		ParString : STRING[260];
	END_STRUCT;
END_TYPE
```

### gES.typ - AutoGen
```iecst
TYPE
	gES_typ : STRUCT
		DIR_MAN_ACTION_ENUM : ARRAY[0..6]OF STRING[32] := ['DIR_MAN_ACTION_NONE', 'DIR_MAN_ACTION_COPY_TO_USER', 'DIR_MAN_ACTION_COPY_TO_USB', 'DIR_MAN_ACTION_DELETE_USER', 'DIR_MAN_ACTION_DELETE_USB', 'DIR_MAN_ACTION_CREATE_DIR_USER', 'DIR_MAN_ACTION_CREATE_DIR_USB'];
		DIR_MAN_STATE_ENUM : ARRAY[0..11]OF STRING[32] := ['DIR_MAN_RESET', 'DIR_MAN_DIRMAKE_CMD', 'DIR_MAN_DIRMAKE_WAIT', 'DIR_MAN_DIRREAD_CMD', 'DIR_MAN_DIRREAD_WAIT', 'DIR_MAN_DIRREAD_USB_CMD', 'DIR_MAN_DIRREAD_USB_WAIT', 'DIR_MAN_DIRSANITIZE_CMD', 'DIR_MAN_DIRSANITIZE_WAIT', 'DIR_MAN_TRANSFER_CMD', 'DIR_MAN_TRANSFER_WAIT', 'DIR_MAN_DELAY'];
		TIME_STATE_ENUM : ARRAY[0..5]OF STRING[32] := ['TIME_RESET_C', 'TIME_CHECKPARREADY_W', 'TIME_IDLE_I', 'TIME_SET_C', 'TIME_SET_W', 'TIME_ERROR'];
		RECIPE_ID_ENUM : ARRAY[0..1]OF STRING[32] := ['RECIPE_ID_REM', 'RECIPE_ID_PAR'];
		MON_ENUM : ARRAY[0..10]OF STRING[32] := ['MON_SYSTEM_PAR_NOT_READY', 'MON_SYSTEM_HMI_STOP', 'MON_SAFETY_ESTOP', 'MON_RECIPE_REM_LOST_REM', 'MON_RECIPE_LOAD_BAD_REM', 'MON_RECIPE_LOAD_GOOD_REM', 'MON_RECIPE_GEN_ERR_REM', 'MON_RECIPE_REM_LOST_PAR', 'MON_RECIPE_LOAD_BAD_PAR', 'MON_RECIPE_LOAD_GOOD_PAR', 'MON_RECIPE_GEN_ERR_PAR'];
		PROCESS_ENUM : ARRAY[0..1]OF STRING[32] := ['PROCESS_MASTER', 'PROCESS_TEMP'];
		MASTER_EVAL_ENUM : ARRAY[0..8]OF STRING[32] := ['MASTER_EVAL_RESET', 'MASTER_EVAL_INIT', 'MASTER_EVAL_STOP_UNCONTROLLED', 'MASTER_EVAL_STOP_CONTROLLED', 'MASTER_EVAL_STOP_NORMAL', 'MASTER_EVAL_UNPAUSE', 'MASTER_EVAL_PAUSE', 'MASTER_EVAL_WAIT_BUFFER_EMPTY', 'MASTER_EVAL_START'];
		MASTER_CALL_ENUM : ARRAY[0..7]OF STRING[32] := ['MASTER_CALL_IDLE', 'MASTER_CALL_RESET', 'MASTER_CALL_STOP_UNCONTROLLED', 'MASTER_CALL_STOP_CONTROLLED', 'MASTER_CALL_STOP_NORMAL', 'MASTER_CALL_UNPAUSE', 'MASTER_CALL_PAUSE', 'MASTER_CALL_START'];
		DRIVER_INST_IN_ENUM : ARRAY[0..0]OF STRING[32] := ['DRIVER_INST_IN_0'];
		C_IN_ENUM : ARRAY[0..8]OF STRING[32] := ['C_IN_RESET', 'C_IN_CLEARCMD', 'C_IN_CLEARMON', 'C_IN_DEFAULTMON', 'C_IN_CLEARPAR', 'C_IN_DEFAULTPAR', 'C_IN_SAVEPAR', 'C_IN_FORCEENABLE', 'C_IN_FORCEDISABLE'];
		M_IN_ENUM : ARRAY[0..0]OF STRING[32] := ['M_IN_DI_ESTOP'];
		W_IN_ENUM : ARRAY[0..0]OF STRING[32] := ['W_IN_DI_ESTOP'];
		DRIVER_INST_DO_ENUM : ARRAY[0..0]OF STRING[32] := ['DRIVER_INST_DO_0'];
		C_DO_ENUM : ARRAY[0..9]OF STRING[32] := ['C_DO_RESET', 'C_DO_CLEARCMD', 'C_DO_CLEARMON', 'C_DO_CLEARPAR', 'C_DO_DEFAULTMON', 'C_DO_DEFAULTPAR', 'C_DO_SAVEPAR', 'C_DO_ERRORRESET', 'C_DO_DISABLEALL', 'C_DO_ENABLE'];
		M_DO_ENUM : ARRAY[0..0]OF STRING[32] := ['M_DO_ERROR'];
		W_DO_ENUM : ARRAY[0..0]OF STRING[32] := ['W_DO_NOERROR'];
		DRIVER_INST_AB_ENUM : ARRAY[0..11]OF STRING[32] := ['DRIVER_INST_AB_VX_0', 'DRIVER_INST_AB_VY_0', 'DRIVER_INST_AB_VZ_0', 'DRIVER_INST_AB_VT_0', 'DRIVER_INST_AB_VV_0', 'DRIVER_INST_AB_RX_0_0', 'DRIVER_INST_AB_RY_0_0', 'DRIVER_INST_AB_RZ_0_0', 'DRIVER_INST_AB_RT_0_0', 'DRIVER_INST_AB_RV_0_0', 'DRIVER_INST_AB_RP_0_0', 'DRIVER_INST_AB_RP_1_0'];
		C_AB_ENUM : ARRAY[0..21]OF STRING[32] := ['C_AB_RESET', 'C_AB_CLEARCMD', 'C_AB_CLEARMON', 'C_AB_DEFAULTMON', 'C_AB_CLEARPAR', 'C_AB_DEFAULTPAR', 'C_AB_SAVEPAR', 'C_AB_LOADPAR', 'C_AB_ERRORRESET', 'C_AB_HOME', 'C_AB_POWER', 'C_AB_UPDATE', 'C_AB_AUTOTUNE', 'C_AB_JOGPOSITIVE', 'C_AB_JOGNEGATIVE', 'C_AB_LIMITLOAD', 'C_AB_STOP', 'C_AB_MOVEABSOLUTE', 'C_AB_MOVEADDITIVE', 'C_AB_MOVEVELOCITY', 'C_AB_RELEASEBRAKE', 'C_AB_SIMULATE'];
		M_AB_ENUM : ARRAY[0..1]OF STRING[32] := ['M_AB_ERROR', 'M_AB_NOTPOWERON'];
		W_AB_ENUM : ARRAY[0..18]OF STRING[32] := ['W_AB_NOERROR', 'W_AB_COMMUNICATIONREADY', 'W_AB_READYTOPOWERON', 'W_AB_POWERON', 'W_AB_ISHOMED', 'W_AB_LIMITLOADACTIVE', 'W_AB_MOVEDONE', 'W_AB_UPDATEDONE', 'W_AB_AUTOTUNEDONE', 'W_AB_BRAKERELEASED', 'W_AB_COMMANDABORTED', 'W_AB_COMMANDBUSY', 'W_AB_INPOSITION', 'W_AB_INVELOCITY', 'W_AB_MOVEACTIVE', 'W_AB_STOPPED', 'W_AB_JOGGING', 'W_AB_JOGLIMITREACHED', 'W_AB_SIMULATION'];
		DRIVER_INST_CS_ENUM : ARRAY[0..9]OF STRING[32] := ['DRIVER_INST_CS_VX_0', 'DRIVER_INST_CS_VY_0', 'DRIVER_INST_CS_VZ_0', 'DRIVER_INST_CS_VT_0', 'DRIVER_INST_CS_VV_0', 'DRIVER_INST_CS_RX_0_0', 'DRIVER_INST_CS_RY_0_0', 'DRIVER_INST_CS_RZ_0_0', 'DRIVER_INST_CS_RT_0_0', 'DRIVER_INST_CS_RV_0_0'];
		C_CS_ENUM : ARRAY[0..13]OF STRING[32] := ['C_CS_RESET', 'C_CS_CLEARCMD', 'C_CS_CLEARMON', 'C_CS_DEFAULTMON', 'C_CS_CLEARPAR', 'C_CS_DEFAULTPAR', 'C_CS_SAVEPAR', 'C_CS_LOADPAR', 'C_CS_ERRORRESET', 'C_CS_MOVECYCLICPOSITION', 'C_CS_MOVECYCLICVELOCITY', 'C_CS_TORQUECONTROL', 'C_CS_TORQUEFEEDFORWARD', 'C_CS_UPDATE'];
		M_CS_ENUM : ARRAY[0..6]OF STRING[32] := ['M_CS_ERROR', 'M_CS_NOTMOVECYCLICPOSITIONACTIVE', 'M_CS_NOTMOVECYCLICVELOCITYACTIVE', 'M_CS_NOTTORQUECONTROLACTIVE', 'M_CS_NOTTORQUEFEEDFORWARDACTIVE', 'M_CS_TCAXISLIMITACTIVE', 'M_CS_NOTTCINTORQUE'];
		W_CS_ENUM : ARRAY[0..12]OF STRING[32] := ['W_CS_NOERROR', 'W_CS_COMMANDABORTED', 'W_CS_COMMANDBUSY', 'W_CS_UPDATEDONE', 'W_CS_MOVECYCLICPOSITIONACTIVE', 'W_CS_MOVECYCLICVELOCITYACTIVE', 'W_CS_TORQUECONTROLACTIVE', 'W_CS_TORQUEFEEDFORWARDACTIVE', 'W_CS_TCAXISLIMITACTIVE', 'W_CS_TCDATAINITIALIZED', 'W_CS_TCINTORQUE', 'W_CS_TCREADY', 'W_CS_AXISREADY'];
		DRIVER_INST_CN_ENUM : ARRAY[0..0]OF STRING[32] := ['DRIVER_INST_CN_0'];
		C_CN_ENUM : ARRAY[0..18]OF STRING[32] := ['C_CN_RESET', 'C_CN_CLEARCMD', 'C_CN_CLEARMON', 'C_CN_DEFAULTMON', 'C_CN_CLEARPAR', 'C_CN_DEFAULTPAR', 'C_CN_SAVEPAR', 'C_CN_LOADPAR', 'C_CN_ERRORRESET', 'C_CN_HOME', 'C_CN_POWER', 'C_CN_UPDATE', 'C_CN_MOVEPROGRAM', 'C_CN_INTERRUPT', 'C_CN_CONTINUE', 'C_CN_STOP', 'C_CN_JOG', 'C_CN_MOVEBLOCK', 'C_CN_SINGLESTEP'];
		M_CN_ENUM : ARRAY[0..2]OF STRING[32] := ['M_CN_ERROR', 'M_CN_NOTPOWERON', 'M_CN_NOTMOVEACTIVE'];
		W_CN_ENUM : ARRAY[0..14]OF STRING[32] := ['W_CN_NOERROR', 'W_CN_COMMUNICATIONREADY', 'W_CN_READYTOPOWERON', 'W_CN_POWERON', 'W_CN_ISHOMED', 'W_CN_WAITFORCONTINUE', 'W_CN_MOVEDONE', 'W_CN_UPDATEDONE', 'W_CN_MOVEINTERRUPTED', 'W_CN_COMMANDABORTED', 'W_CN_COMMANDBUSY', 'W_CN_INMOTION', 'W_CN_MOVEACTIVE', 'W_CN_STOPPED', 'W_CN_SINGLESTEPACTIVE'];
		DRIVER_INST_TR_ENUM : ARRAY[0..0]OF STRING[32] := ['DRIVER_INST_TR_0'];
		C_TR_ENUM : ARRAY[0..10]OF STRING[32] := ['C_TR_RESET', 'C_TR_CLEARCMD', 'C_TR_CLEARMON', 'C_TR_DEFAULTMON', 'C_TR_CLEARPAR', 'C_TR_DEFAULTPAR', 'C_TR_SAVEPAR', 'C_TR_LOADPAR', 'C_TR_ERRORRESET', 'C_TR_ENABLE', 'C_TR_RESYNC'];
		M_TR_ENUM : ARRAY[0..0]OF STRING[32] := ['M_TR_ERROR'];
		W_TR_ENUM : ARRAY[0..0]OF STRING[32] := ['W_TR_NOERROR'];
		DRIVER_INST_MR_ENUM : ARRAY[0..0]OF STRING[32] := ['DRIVER_INST_MR_0'];
		C_MR_ENUM : ARRAY[0..12]OF STRING[32] := ['C_MR_RESET', 'C_MR_CLEARCMD', 'C_MR_CLEARMON', 'C_MR_DEFAULTMON', 'C_MR_CLEARPAR', 'C_MR_DEFAULTPAR', 'C_MR_SAVEPAR', 'C_MR_LOADPAR', 'C_MR_ERRORRESET', 'C_MR_MBMOPEN', 'C_MR_MBMASTER', 'C_MR_MBMCLOSE', 'C_MR_MBMCMD'];
		M_MR_ENUM : ARRAY[0..0]OF STRING[32] := ['M_MR_ERROR'];
		W_MR_ENUM : ARRAY[0..4]OF STRING[32] := ['W_MR_NOERROR', 'W_MR_MBMOPEN', 'W_MR_MBMASTER', 'W_MR_MBMCLOSE', 'W_MR_MBMCMD'];
		DRIVER_INST_BX_ENUM : ARRAY[0..0]OF STRING[32] := ['DRIVER_INST_BX_0'];
		C_BX_ENUM : ARRAY[0..9]OF STRING[32] := ['C_BX_RESET', 'C_BX_CLEARCMD', 'C_BX_CLEARMON', 'C_BX_DEFAULTMON', 'C_BX_CLEARPAR', 'C_BX_DEFAULTPAR', 'C_BX_SAVEPAR', 'C_BX_LOADPAR', 'C_BX_ERRORRESET', 'C_BX_ENABLE'];
		M_BX_ENUM : ARRAY[0..0]OF STRING[32] := ['M_BX_ERROR'];
		W_BX_ENUM : ARRAY[0..1]OF STRING[32] := ['W_BX_NOERROR', 'W_BX_ACTIVE'];
	END_STRUCT;
END_TYPE
```

### Package Logical/Libraries - Global libraries

### Data object Logical/Libraries/AcpParTabL (Apt)

#### AcpParTabL.apt - ACOPOS Parameter table
```
AcoposParameterTable:
  Root Parameters:
    728 = 2 (Name=ENCOD2_LINE_CHK_IGNORE)  // Encoder2: Ignore check
```

### Data object Logical/Libraries/MbRTU (Simple)

#### MbRTU.dat
```
;--------------------
; Modbus command file
;--------------------
"gIO.VFD[0].EventRead[00]       ", 03, $01, "gIO.VFD[0].DataRead[00]        ", 8603, 0001
"gIO.VFD[0].EventRead[01]       ", 03, $01, "gIO.VFD[0].DataRead[01]        ", 8604, 0001
"gIO.VFD[0].EventRead[02]       ", 03, $01, "gIO.VFD[0].DataRead[02]        ", 7121, 0001
"gIO.VFD[0].EventWrite[00]      ", 06, $01, "gIO.VFD[0].DataWrite[00]       ", 8601, 0001
"gIO.VFD[0].EventWrite[01]      ", 06, $01, "gIO.VFD[0].DataWrite[01]       ", 8602, 0001
"gIO.VFD[1].EventRead[00]       ", 03, $02, "gIO.VFD[1].DataRead[00]        ", 8603, 0001
"gIO.VFD[1].EventRead[01]       ", 03, $02, "gIO.VFD[1].DataRead[01]        ", 8604, 0001
"gIO.VFD[1].EventRead[02]       ", 03, $02, "gIO.VFD[1].DataRead[02]        ", 7121, 0001
"gIO.VFD[1].EventWrite[00]      ", 06, $02, "gIO.VFD[1].DataWrite[00]       ", 8601, 0001
"gIO.VFD[1].EventWrite[01]      ", 06, $02, "gIO.VFD[1].DataWrite[01]       ", 8602, 0001

;"gIO.VFD.EventRead[00]          ", 03, $01, "gIO.VFD.DataRead[00]           ", 0000, 0001
;"gIO.VFD.EventWrite[00]         ", 06, $01, "gIO.VFD.DataWrite[00]          ", 0000, 0001
; \_____________________________/	|    |    \_____________________________/    |      |
;			 	 |					|    |				  	 |				     |      |
;		   31 Characters		    |    |			   31 Characters  		     |      |_Number of coils or registers
;			 						|    |				   						 |_Offset of the Modbus Variables
;									|    |
;									|    |_Target Address of the slave station
;			 						|
;			 						|_ Modbus function

; 01 Read coil status
; 02 Read input status
; 03 Read holding register
; 04 Read input register
; 05 Force single coil
; 06 Preset single register
; 15 Force multiple coils
; 16 Preset multiple registers
```

- Project.language (not shown)

### Library Logical/Libraries/TC_General (IEC)

#### Types.typ - Exported data types
```iecst
TYPE
	TC_TypeSelect_typ : 	STRUCT
		Select : TC_TYPE_ENUM;
		VarSINT : SINT;
		VarUSINT : USINT;
		VarINT : INT;
		VarUINT : UINT;
		VarDINT : DINT;
		VarUDINT : UDINT;
		VarREAL : REAL;
		VarLREAL : LREAL;
		VarTIME : TIME;
		VarDT : DATE_AND_TIME;
		VarSTRING_ADR : UDINT;
		VarSTRING_LEN : UDINT;
		VarWSTRING_ADR : UDINT;
		VarWSTRING_LEN : UDINT;
	END_STRUCT;
	TC_TYPE_ENUM :
		(
		TC_TYPE_INT,
		TC_TYPE_USINT,
		TC_TYPE_SINT,
		TC_TYPE_UINT,
		TC_TYPE_DINT,
		TC_TYPE_UDINT,
		TC_TYPE_REAL,
		TC_TYPE_LREAL,
		TC_TYPE_TIME,
		TC_TYPE_DT,
		TC_TYPE_STRING,
		TC_TYPE_WSTRING
		);
END_TYPE
```

### Library Logical/Libraries/TC_Version (IEC, version 1.0.0)
Depends on: ArEventLog, ArProject, AsBrStr

#### IdentifyConfig.st
```iecst
(* returns the ID and Version of the configuration as strings and also enters a record in the log book *)
FUNCTION_BLOCK IdentifyConfig
	Done := FALSE;
	CASE internal.state OF
		0:
			IF internal.ArProjectGetInfo_0.Done THEN
				ConfigID := internal.ArProjectGetInfo_0.ConfigurationID;
				ConfigVersion := internal.ArProjectGetInfo_0.ConfigurationVersion;
				internal.AddData := '';
				brsstrcat(ADR(internal.AddData),ADR('Configuration ID="'));
				brsstrcat(ADR(internal.AddData),ADR(ConfigID));
				brsstrcat(ADR(internal.AddData),ADR('" Configuration version="'));
				brsstrcat(ADR(internal.AddData),ADR(ConfigVersion));
				brsstrcat(ADR(internal.AddData),ADR('"'));
				internal.ArProjectGetInfo_0.Execute := FALSE;
				internal.state := 10;
			ELSIF NOT internal.ArProjectGetInfo_0.Execute THEN
				internal.ArProjectGetInfo_0.Execute := TRUE;
			ELSE
				internal.ArProjectGetInfo_0.Execute := FALSE;
			END_IF;
		10:
			IF internal.ArEventLogGetIdent_0.Done THEN
				internal.ArEventLogGetIdent_0.Execute := FALSE;
				internal.ArEventLogWrite_0.Ident := internal.ArEventLogGetIdent_0.Ident;
				internal.ArEventLogWrite_0.EventID := 1610612736;
				internal.ArEventLogWrite_0.ObjectID := 'TC_Version';
				internal.ArEventLogWrite_0.AddDataFormat := 1;
				internal.ArEventLogWrite_0.AddData := ADR(internal.AddData);
				internal.ArEventLogWrite_0.AddDataSize := brsstrlen(ADR(internal.AddData))+1;
				internal.ArEventLogWrite_0.Execute := TRUE;
				internal.state := 20;
			ELSIF NOT internal.ArEventLogGetIdent_0.Execute THEN
				internal.ArEventLogGetIdent_0.Name := '$$arlogusr';
				internal.ArEventLogGetIdent_0.Execute := TRUE;
			ELSE
				internal.ArEventLogGetIdent_0.Execute := FALSE;
			END_IF;
		20:
			IF internal.ArEventLogWrite_0.Done THEN
				internal.ArEventLogWrite_0.Execute := FALSE;
				internal.state := 30;
			ELSIF NOT internal.ArEventLogWrite_0.Execute THEN
				internal.ArEventLogWrite_0.Execute := TRUE;
			ELSE
				internal.ArEventLogWrite_0.Execute := FALSE;
			END_IF;
		30:
			Done := TRUE;
	END_CASE;

	internal.ArProjectGetInfo_0();
	internal.ArEventLogGetIdent_0();
	internal.ArEventLogWrite_0();

END_FUNCTION_BLOCK
```

### Library Logical/Libraries/TC_IO (IEC)

#### Types.typ - Exported data types
```iecst
TYPE
	TC_IO_Digital_Sim_typ : 	STRUCT
		Active : BOOL;
		Logical : BOOL;
	END_STRUCT;
	TC_IO_Digital_Signal_typ : 	STRUCT
		Logical : BOOL;
		EdgePosLogical : BOOL;
		EdgeNegLogical : BOOL;
		Filtered : BOOL;
		EdgePosFiltered : BOOL;
		EdgeNegFiltered : BOOL;
		IOMapping : BOOL;
		InvertedIOMapping : BOOL;
		VisIOMapping : BOOL;
		VisRefresher : BOOL;
	END_STRUCT;
	TC_IO_Digital_Par_LimitSet_typ : 	STRUCT
		FilterOnTime_Min : LREAL;
		FilterOnTime_Max : LREAL;
		FilterOffTime_Min : LREAL;
		FilterOffTime_Max : LREAL;
	END_STRUCT;
	TC_IO_Digital_Par_typ : 	STRUCT
		InvertedIOMapping : BOOL;
		FilterOnTime : LREAL;
		FilterOffTime : LREAL;
	END_STRUCT;
	TC_IO_Digital_Internal_typ : 	STRUCT
		StatusLogical : BOOL;
		StatusFiltered : BOOL;
		CTON_DB_Off : CTON;
		CTON_DB_On : CTON;
	END_STRUCT;
	TC_IO_Digital_Forcing_typ : 	STRUCT
		Off : BOOL;
		On : BOOL;
	END_STRUCT;
	TC_IO_Analog_Sim_typ : 	STRUCT
		Active : BOOL;
		Logical : LREAL;
	END_STRUCT;
	TC_IO_Analog_Signal_typ : 	STRUCT
		UnlimitedLogical : LREAL;
		MinExceeded : BOOL;
		MaxExceeded : BOOL;
		Logical : LREAL;
		Filtered : LREAL;
		Vis : TC_IO_Analog_Vis_typ;
		IOMapping : TC_IO_Analog_Mapping_typ;
	END_STRUCT;
	TC_IO_Analog_Par_LimitSet_typ : 	STRUCT
		M_Min : LREAL;
		M_Max : LREAL;
		B_Min : LREAL;
		B_Max : LREAL;
		Filter_Min : LREAL;
		Filter_Max : LREAL;
		MinValue_Min : LREAL;
		MinValue_Max : LREAL;
		MaxValue_Min : LREAL;
		MaxValue_Max : LREAL;
	END_STRUCT;
	TC_IO_Analog_Par_typ : 	STRUCT
		M : LREAL;
		B : LREAL;
		Filter : LREAL;
		MaxValue : LREAL;
		MinValue : LREAL;
	END_STRUCT;
	TC_IO_Analog_Internal_typ : 	STRUCT
		InitFilter : BOOL;
		Filter : LREAL;
		LastFilter : LREAL;
		Temp : LREAL;
	END_STRUCT;
	TC_IO_Analog_Forcing_typ : 	STRUCT
		Off : BOOL;
		On : BOOL;
		Value : LREAL;
	END_STRUCT;
	TC_IO_Analog_Vis_typ : 	STRUCT
		Raw : LREAL;
		IO : LREAL;
		App : LREAL;
	END_STRUCT;
	TC_IO_Analog_Mapping_typ : 	STRUCT
		VarSINT : SINT;
		VarUSINT : USINT;
		VarINT : INT;
		VarUINT : UINT;
		VarDINT : DINT;
		VarUDINT : UDINT;
		VarREAL : REAL;
		VarLREAL : LREAL;
	END_STRUCT;
	TC_IO_ANALOG_TYPE_ENUM :
		(
		TC_IO_ANALOG_TYPE_INT,
		TC_IO_ANALOG_TYPE_USINT,
		TC_IO_ANALOG_TYPE_SINT,
		TC_IO_ANALOG_TYPE_UINT,
		TC_IO_ANALOG_TYPE_DINT,
		TC_IO_ANALOG_TYPE_UDINT,
		TC_IO_ANALOG_TYPE_REAL,
		TC_IO_ANALOG_TYPE_LREAL
		);
END_TYPE
```

#### TC_IO.fun - Exported functions and function blocks
```iecst
{REDUND_ERROR} FUNCTION_BLOCK TC_IO_DO (* *) (*$GROUP=User,$CAT=User,$GROUPICON=User.png,$CATICON=User.png*)
	VAR_INPUT
		Logical : BOOL;
		Forcing : TC_IO_Digital_Forcing_typ;
		Par : TC_IO_Digital_Par_typ;
	END_VAR
	VAR_OUTPUT
		Signal : TC_IO_Digital_Signal_typ;
	END_VAR
	VAR
		Internal : TC_IO_Digital_Internal_typ;
	END_VAR
END_FUNCTION_BLOCK

{REDUND_ERROR} FUNCTION_BLOCK TC_IO_DI (* *) (*$GROUP=User,$CAT=User,$GROUPICON=User.png,$CATICON=User.png*)
	VAR_INPUT
		IOMapping : BOOL;
		Forcing : TC_IO_Digital_Forcing_typ;
		Par : TC_IO_Digital_Par_typ;
		Sim : TC_IO_Digital_Sim_typ;
	END_VAR
	VAR_OUTPUT
		Signal : TC_IO_Digital_Signal_typ;
	END_VAR
	VAR
		Internal : TC_IO_Digital_Internal_typ;
	END_VAR
END_FUNCTION_BLOCK

{REDUND_ERROR} FUNCTION_BLOCK TC_IO_AI (* *) (*$GROUP=User,$CAT=User,$GROUPICON=User.png,$CATICON=User.png*)
	VAR_INPUT
		VarType : TC_IO_ANALOG_TYPE_ENUM;
		IOMapping : TC_IO_Analog_Mapping_typ;
		Forcing : TC_IO_Analog_Forcing_typ;
		Sim : TC_IO_Analog_Sim_typ;
		Par : TC_IO_Analog_Par_typ;
	END_VAR
	VAR_OUTPUT
		Signal : TC_IO_Analog_Signal_typ;
	END_VAR
	VAR
		Internal : TC_IO_Analog_Internal_typ;
	END_VAR
END_FUNCTION_BLOCK

{REDUND_ERROR} FUNCTION_BLOCK TC_IO_AO (* *) (*$GROUP=User,$CAT=User,$GROUPICON=User.png,$CATICON=User.png*)
	VAR_INPUT
		VarType : TC_IO_ANALOG_TYPE_ENUM;
		Logical : LREAL;
		Forcing : TC_IO_Analog_Forcing_typ;
		Par : TC_IO_Analog_Par_typ;
	END_VAR
	VAR_OUTPUT
		Signal : TC_IO_Analog_Signal_typ;
	END_VAR
	VAR
		Internal : TC_IO_Analog_Internal_typ;
	END_VAR
END_FUNCTION_BLOCK
```

#### TC_IO_DI.st
```iecst
(* Full Digital Input Handler*)
FUNCTION_BLOCK TC_IO_DI

//LOGICAL/INVERT
	Signal.IOMapping					:= IOMapping;
	Signal.InvertedIOMapping			:= NOT Signal.IOMapping;
	IF Par.InvertedIOMapping THEN
		Signal.Logical					:= Signal.InvertedIOMapping;
	ELSE
		Signal.Logical					:= Signal.IOMapping;
	END_IF;
//SIMULATION
	IF Sim.Active THEN
		Signal.Logical					:= Sim.Logical;
		Signal.IOMapping				:= Sim.Logical;
		Signal.InvertedIOMapping		:= NOT Sim.Logical;
	END_IF;
//VISUALIZATION
	IF Par.InvertedIOMapping THEN
		Signal.VisIOMapping				:= Signal.InvertedIOMapping;
	ELSE
		Signal.VisIOMapping				:= Signal.IOMapping;
	END_IF;
//DEBOUNCING
	IF Signal.Logical THEN
		Internal.CTON_DB_Off(IN := FALSE);
		IF Internal.CTON_DB_On.Q OR Par.FilterOnTime <= 0.0 THEN
			Signal.Filtered			:= TRUE;
		ELSE
			Internal.CTON_DB_On(IN := TRUE, PT := LREAL_TO_TIME(Par.FilterOnTime*1000.0));
		END_IF;
	ELSE
		Internal.CTON_DB_On(IN := FALSE);
		IF Internal.CTON_DB_Off.Q OR Par.FilterOffTime <= 0.0 THEN
			Signal.Filtered			:= FALSE;
		ELSE
			Internal.CTON_DB_Off(IN := TRUE, PT := LREAL_TO_TIME(Par.FilterOffTime*1000.0));
		END_IF;
	END_IF;
//FORCING
	IF Forcing.On XOR Forcing.Off THEN
		IF Forcing.Off THEN
			Signal.Logical				:= FALSE;
			Signal.Filtered			:= FALSE;
		ELSIF Forcing.On THEN
			Signal.Logical				:= TRUE;
			Signal.Filtered			:= TRUE;
		END_IF;
	END_IF;
//EDGES
	Signal.EdgeNegLogical				:= FALSE;
	IF Internal.StatusLogical AND NOT Signal.Logical THEN
		Signal.EdgeNegLogical			:= TRUE;
	END_IF;
	Signal.EdgePosLogical				:= FALSE;
	IF NOT Internal.StatusLogical AND Signal.Logical THEN
		Signal.EdgePosLogical			:= TRUE;
	END_IF;
	Internal.StatusLogical 				:= Signal.Logical;

	Signal.EdgeNegFiltered				:= FALSE;
	IF Internal.StatusFiltered AND NOT Signal.Filtered THEN
		Signal.EdgeNegFiltered			:= TRUE;
	END_IF;
	Signal.EdgePosFiltered				:= FALSE;
	IF NOT Internal.StatusFiltered AND Signal.Filtered THEN
		Signal.EdgePosFiltered			:= TRUE;
	END_IF;
	Internal.StatusFiltered 			:= Signal.Filtered;

//This is needed as a workaround for an event bug that wouldnt show IO status colors if IO was active at start of Vis
	Signal.VisRefresher					:= FALSE;

END_FUNCTION_BLOCK
```

#### TC_IO_DO.st
```iecst
(* Full Digital Output Handler*)
FUNCTION_BLOCK TC_IO_DO

//LOGICAL
	Signal.Logical						:= Logical;
//DEBOUNCING
	IF Signal.Logical THEN
		Internal.CTON_DB_Off(IN := FALSE);
		IF Internal.CTON_DB_On.Q OR Par.FilterOnTime <= 0.0 THEN
			Signal.Filtered			:= TRUE;
		ELSE
			Internal.CTON_DB_On(IN := TRUE, PT := LREAL_TO_TIME(Par.FilterOnTime*1000.0));
		END_IF;
	ELSE
		Internal.CTON_DB_On(IN := FALSE);
		IF Internal.CTON_DB_Off.Q OR Par.FilterOffTime <= 0.0 THEN
			Signal.Filtered			:= FALSE;
		ELSE
			Internal.CTON_DB_Off(IN := TRUE, PT := LREAL_TO_TIME(Par.FilterOffTime*1000.0));
		END_IF;
	END_IF;
//EDGES
	Signal.EdgeNegLogical				:= FALSE;
	IF Internal.StatusLogical AND NOT Signal.Logical THEN
		Signal.EdgeNegLogical			:= TRUE;
	END_IF;
	Signal.EdgePosLogical				:= FALSE;
	IF NOT Internal.StatusLogical AND Signal.Logical THEN
		Signal.EdgePosLogical			:= TRUE;
	END_IF;
	Internal.StatusLogical 				:= Signal.Logical;

	Signal.EdgeNegFiltered				:= FALSE;
	IF Internal.StatusFiltered AND NOT Signal.Filtered THEN
		Signal.EdgeNegFiltered			:= TRUE;
	END_IF;
	Signal.EdgePosFiltered				:= FALSE;
	IF NOT Internal.StatusFiltered AND Signal.Filtered THEN
		Signal.EdgePosFiltered			:= TRUE;
	END_IF;
	Internal.StatusFiltered 			:= Signal.Filtered;
//FORCING
	Signal.IOMapping					:= Signal.Filtered;
	IF Forcing.On XOR Forcing.Off THEN
		IF Forcing.Off THEN
			Signal.IOMapping			:= FALSE;
		ELSIF Forcing.On THEN
			Signal.IOMapping			:= TRUE;
		END_IF;
	END_IF;
//INVERT
	Signal.InvertedIOMapping			:= NOT Signal.IOMapping;
//VISUALIZATION
	IF Par.InvertedIOMapping THEN
		Signal.VisIOMapping				:= Signal.InvertedIOMapping;
	ELSE
		Signal.VisIOMapping				:= Signal.IOMapping;
	END_IF;

//This is needed as a workaround for an event bug that wouldnt show IO status colors if IO was active at start of Vis
	Signal.VisRefresher					:= FALSE;

END_FUNCTION_BLOCK
```

#### TC_IO_AO.st
```iecst
(* Full Analog Output Handler*)
FUNCTION_BLOCK TC_IO_AO
//LOGICAL
	Signal.Logical						:= Logical;
	Signal.UnlimitedLogical				:= Logical;
	Signal.Vis.App						:= Logical;
	Internal.Temp						:= Logical;
//FORCING
	IF Forcing.On XOR Forcing.Off THEN
		IF Forcing.Off THEN
			Internal.Temp				:= 0.0;
		ELSIF Forcing.On THEN
			Internal.Temp				:= Forcing.Value;
		END_IF;
	END_IF;
//LIMITING
	Signal.MaxExceeded					:= FALSE;
	IF Internal.Temp > Par.MaxValue THEN
		Signal.MaxExceeded				:= TRUE;
		Internal.Temp					:= Par.MaxValue;
	END_IF;
	Signal.MinExceeded					:= FALSE;
	IF Signal.Logical < Par.MinValue THEN
		Signal.MinExceeded				:= TRUE;
		Internal.Temp					:= Par.MinValue;
	END_IF;
//FILTERING
	Internal.Filter 					:= Par.Filter;
	IF Par.Filter < 0.0 THEN
		Internal.Filter 				:= 0.0;
	ELSIF Internal.Filter > 1.0 THEN
		Internal.Filter 				:= 0.99999999;
	END_IF;
	IF NOT Internal.InitFilter OR Internal.LastFilter <> Internal.Filter THEN
		Internal.InitFilter				:= TRUE;
		Internal.LastFilter 			:= Internal.Filter;
		Signal.Filtered 				:= Internal.Temp;
	ELSE
		Signal.Filtered 				:= Internal.Temp*(1.0-Internal.Filter) + Signal.Filtered*Internal.Filter;
	END_IF;
	IF Signal.Filtered > Par.MaxValue THEN
		Signal.Filtered 				:= Par.MaxValue;
	ELSIF Signal.Filtered < Par.MinValue THEN
		Signal.Filtered 				:= Par.MinValue;
	END_IF;
//IOMAPPING
	Signal.Vis.IO						:= Signal.Filtered;
	IF Par.M <> 0 THEN
		Signal.Vis.Raw		 			:= (Signal.Filtered-Par.B)/Par.M;
	ELSE
		Signal.Vis.Raw 					:= 0.0;
	END_IF;
	CASE VarType OF
		TC_IO_ANALOG_TYPE_INT:
			Signal.IOMapping.VarINT		:= LREAL_TO_INT(Signal.Vis.Raw);
		TC_IO_ANALOG_TYPE_USINT:
			Signal.IOMapping.VarUSINT	:= LREAL_TO_USINT(Signal.Vis.Raw);
		TC_IO_ANALOG_TYPE_SINT:
			Signal.IOMapping.VarSINT	:= LREAL_TO_SINT(Signal.Vis.Raw);
		TC_IO_ANALOG_TYPE_UINT:
			Signal.IOMapping.VarUINT	:= LREAL_TO_UINT(Signal.Vis.Raw);
		TC_IO_ANALOG_TYPE_DINT:
			Signal.IOMapping.VarDINT	:= LREAL_TO_DINT(Signal.Vis.Raw);
		TC_IO_ANALOG_TYPE_UDINT:
			Signal.IOMapping.VarUDINT	:= LREAL_TO_UDINT(Signal.Vis.Raw);
		TC_IO_ANALOG_TYPE_REAL:
			Signal.IOMapping.VarREAL	:= LREAL_TO_REAL(Signal.Vis.Raw);
		TC_IO_ANALOG_TYPE_LREAL:
			Signal.IOMapping.VarLREAL	:= Signal.Vis.Raw;
	END_CASE

END_FUNCTION_BLOCK
```
